32 Dword FIFO memory
*)
IF rst THEN
	(* asynchronous reset for the fifo *)
	NW := 0;
	NR := 0;
	Dout := 0;
	empty := TRUE;
	full := FALSE;
ELSIF WR AND E AND NOT full THEN
	(* write action *)
	fifo[NW] := Din;
	IF NW = top THEN NW := 0; ELSE NW := NW + 1; END_IF;
	full := NW = NR;
	empty := FALSE;
ELSIF NOT WR AND E AND NOT empty THEN
	(* read from stack *)
	Dout := fifo[NR];
	IF NR = top THEN NR := 0; ELSE NR := NR + 1; END_IF;
	empty := NR = NW;
	full := FALSE;
END_IF;

(* revision history
hm		4. aug. 2006	rev 1.0
	original version

hm		19. feb 2008	rev 1.1
	performance improvements

*)
END_FUNCTION_BLOCK

(* POU Logic/memory/STACK_16, ST *)
FUNCTION_BLOCK STACK_16
VAR_INPUT
	Din : DWORD;
	RW : BOOL;
	E : BOOL;
	RST : BOOL;
END_VAR
VAR_OUTPUT
	Dout : DWORD := 0;
	empty : BOOL := TRUE;
	full : BOOL := FALSE;
END_VAR
VAR
	Stack : ARRAY[0..15] OF DWORD;
	N : INT := -1;
	top : INT := 15;
END_VAR

(*
	version 1.1	19 feb 2008
	programmer 	hugo
	tested by		tobias

16 Dword STACK memory
*)
IF rst THEN
	(* asynchronous reset for the fifo *)
	N := -1;
	Dout := 0;
	empty := TRUE;
	full := FALSE;
ELSIF RW AND E AND NOT full THEN
	(* write action *)
	N := N + 1;
	full := N = TOP;
	empty := FALSE;
	stack[N] := Din;
ELSIF NOT RW AND E AND NOT empty THEN
	(* read from stack *)
	Dout := stack[N];
	N := N -1;
	empty := N < 0;
	full := FALSE;
END_IF;


(* revision history
hm		4. aug. 2006	rev 1.0
	original version

hm		19. feb 2008	rev 1.1
	performance improvements

*)
END_FUNCTION_BLOCK

(* POU Logic/memory/STACK_32, ST *)
FUNCTION_BLOCK STACK_32
VAR_INPUT
	Din : DWORD;
	RW : BOOL;
	E : BOOL;
	RST : BOOL;
END_VAR
VAR_OUTPUT
	Dout : DWORD := 0;
	empty : BOOL := TRUE;
	full : BOOL := FALSE;
END_VAR
VAR
	Stack : ARRAY[0..31] OF DWORD;
	N : INT := -1;
	top : INT := 31;
END_VAR

(*
	version 1.1	19. feb 2008
	programmer 	hugo
	tested by		tobias

32 Dword STACK memory
*)
IF rst THEN
	(* asynchronous reset for the fifo *)
	N := -1;
	Dout := 0;
	empty := TRUE;
	full := FALSE;
ELSIF RW AND E AND NOT full THEN
	(* write action *)
	N := N + 1;
	full := N = TOP;
	empty := FALSE;
	stack[N] := Din;
ELSIF NOT RW AND E AND NOT empty THEN
	(* read from stack *)
	Dout := stack[N];
	N := N -1;
	empty := N < 0;
	full := FALSE;
END_IF;


(* revision history
hm		4. aug. 2006	rev 1.0
	original version

hm		19. feb 2008	rev 1.1
	performance improvements

*)
END_FUNCTION_BLOCK

(* POU Logic/Others/matrix, ST *)
FUNCTION_BLOCK matrix
VAR_INPUT
	x1, x2, x3, x4, X5 : BOOL;
END_VAR
VAR_INPUT CONSTANT
	Release : BOOL;
END_VAR
VAR_OUTPUT
	code : BYTE;
	TP : BOOL;
	y1: BOOL := TRUE;
	y2, y3, y4 : BOOL;
END_VAR
VAR
	line : BYTE := 1;
	X : ARRAY[1..4] OF BYTE; (* scan line inputs *)
	L : ARRAY[1..4] OF BYTE; (* scan line status *)
	i: INT;
	temp: BYTE;
END_VAR

(*
version 1.2	23 dec 2007
programmer 	hugo
tested by		tobias

MATRIX is a matrix keyboard encoder for 4 rows and up to 5 columns.
matrix can send a code while a key is pressed and it sends another code while a key is released when the setup variable 'release' is set to true.
the setup variable release is false the code is only sent when the key is pressed.
the output byte holds the 5 columns in the lowest bits 0..2  and the row number in bits 4..6, while bit 7 is true for a key pressed and false for a key released.

*)
TP := FALSE;
code := 0;

(* read scan lines *)
X[line].0 := X1;
X[line].1 := X2;
X[line].2 := X3;
X[line].3 := X4;
X[line].4 := X5;

(* compare for change *)
FOR i := 1 TO 4 DO
	IF X[i] <> L[i] THEN
		(* scan line information has changed code need to be found and generated *)
		temp := x[i] XOR L[i];
		IF temp.0 THEN
			code := 1;
			code.7 := X[i].0;
			L[i].0 := X[i].0;
		ELSIF temp.1 THEN
			code := 2;
			code.7 := X[i].1;
			L[i].1 := X[i].1;
		ELSIF temp.2 THEN
			code := 3;
			code.7 := X[i].2;
			L[i].2 := X[i].2;
		ELSIF temp.3 THEN
			code := 4;
			code.7 := X[i].3;
			L[i].3 := X[i].3;
		ELSIF temp.4 THEN
			code := 5;
			code.7 := X[i].4;
			L[i].4 := X[i].4;
		END_IF;
		TP := TRUE;
		Code.4 := Line.0;
		Code.5 := Line.1;
		Code.6 := Line.2;

		(* check if release codes need to be killed *)
		IF NOT release AND code < 127 THEN
			code := 0;
			TP := 0;
		END_IF;
		EXIT;
	END_IF;
END_FOR;

(* increment scan line every cycle *)
CASE line OF
	1 :	Line := 2;
		Y1 := FALSE; Y3 := FALSE; Y4 := FALSE; Y2 := TRUE;
	2 :	Line := 3;
		Y1 := FALSE; Y2 := FALSE; Y4 := FALSE; Y3 := TRUE;
	3 :	Line := 4;
		Y1 := FALSE; Y2 := FALSE; Y3 := FALSE; Y4 := TRUE;
	4 :	Line := 1;
		Y2 := FALSE; Y3 := FALSE; Y4 := FALSE; Y1 := TRUE;
END_CASE;

(* revision history
hm		10.6.2007	rev 1.0		
	original version 


hm		11.9.2007	rev 1.1		
	deleted unused variables k and old_code

hm		23.12.2007	rev 1.2
	added exit statement in for loop instead of i:=5

*)
END_FUNCTION_BLOCK

(* POU mathematical/functions/FT_avg, ST *)
FUNCTION_BLOCK FT_avg
VAR_INPUT
	in : REAL;
	en : BOOL;
	N : INT;
	rst : BOOL;
END_VAR
VAR_OUTPUT
	avg : REAL;
END_VAR
VAR
	buff : delay;
	i: INT;
	init : BOOL;
END_VAR

(*
version 1.1	7 jan 2007
programmer 	hugo
tested by		tobias

this function calculates the average over n samples from a sequential input
the input values are shifted into an N deep buffer and the avg of this buffer is diplayed at anytime on the output.
a rst will load the buffer with the current in value..

*)
(* limit n to a max of 32 because delay can do max 32 cycles *)
IF N > 32 THEN
	buff.n := 32;
ELSIF N < 0 THEN
	Buff.n := 0;
ELSE
	buff.n := N;
END_IF;

IF NOT init THEN
	FOR i := 1 TO N DO
		buff(in := in);
	END_FOR;
	avg := in;
	init := TRUE;
ELSIF rst THEN
	FOR i := 1 TO N DO
		buff(in := in);
	END_FOR;
	avg := in;
ELSIF en THEN
	buff(in := in);
	avg := avg + (in - buff.out)/N;
END_IF;

(* revision history

hm	7.1.2007	rev 1.1
	chaged rst logic to load the buffer with the actual input value instead of 0.
	added en input to allow better control of signal flow
	added init to load the buffer with in at startup to avoid rampup at beginning.
	deleted unused variable cnt.
*)
END_FUNCTION_BLOCK

(* POU mathematical/functions/FT_min_max, ST *)
FUNCTION_BLOCK FT_min_max
VAR_INPUT
	in : REAL;
	rst : BOOL;
END_VAR
VAR_OUTPUT
	mx : REAL;
	mn : REAL;
END_VAR
VAR
	init: BOOL;
END_VAR

(*
version 1.0	1 sep 2006
programmer 	hugo
tested by		tobias

this function block stores the min and max value of an input signal.
when rst is true the mn and mx outputs are set to the in value.
when a rst is never active the function autoresets to the in value at startup.
since the input might not be present at first cycle the mn and mx are set during second cycle.

*)
IF rst OR NOT init THEN
	mn := in;
	mx := in;
	init := 1;
ELSIF in < mn THEN mn := in;
ELSIF in > mx THEN mx := in;
END_IF;
END_FUNCTION_BLOCK

(* POU Time&Date/Ltime, ST *)
FUNCTION_BLOCK Ltime
VAR_INPUT
	UTC : DT;
	dst_enable : BOOL;
	time_zone_offset : INT;
END_VAR
VAR_OUTPUT
	local_DT : DT;
	DST_on : BOOL;
	wday : INT;
END_VAR
VAR
	tx: TIME;
END_VAR

(*

version 1.6	8 dec 2007
programmer 	oscat
tested by		tobias

ltime is a real time clock that uses the system rtc as utc time and calculates and given time zone.
the utc time is supplied on the input UTC.
according to the input variable time_zone_offset when the input dst_enable is true,
the dst on and off times are calculated by a formula for any given year and the time is advanced and reset by one hour
at 02:00 and 03:00 for the last sunday of march and last sunday of october.
the code is high performance and the rtc counts every second.
if more then one time zone is needed by the systen the clock can be started many times by placing more then one function block.

execution time on wago 750-841 = 20 us 
 
*)
tx := DWORD_TO_TIME(INT_TO_DWORD(ABS(time_zone_offset))* 3600000);
DST_ON := DST(UTC) AND dst_enable;
IF DST_ON THEN
	IF time_zone_offset < 0 THEN local_DT := UTC - tx + t#1h; ELSE local_DT := UTC + tx + t#1h; END_IF;
ELSE
	IF time_zone_offset < 0 THEN local_DT := UTC - tx; ELSE local_DT := UTC + tx; END_IF;
END_IF;
wday := weekday(DT_TO_DATE(local_DT));


(* revision history

hm 2.10.2006	rev 1.1
	corrected an error where dst would be delayed by 0.1second

hm 17.1.2007	rev 1.2
	added utc input instead of internal sysrtcgettime because this would only work on wago.
	dst_enable would not be checked before dst would be enabled.

hm 18.3.2007	rev 1.3
	changed code, dst would not work during first cycle.

hm 24.10.2007	rev 1.4
	changed code because the execution every 100ms can cause major problems if the supplied time was not correct at start.
	use of new dst function

hm 12. nov 2007	rev 1.5
		changed Type of time_zone_offset from time to int to allow for time zones with negative offset

8 dec 2007		rev 1.6
	corrected a problem with time_zone_offset
*)
END_FUNCTION_BLOCK

(* POU XTEST/Performance Test/fc_list, ST *)
FUNCTION_BLOCK fc_list
VAR_INPUT
	num : INT;
	check : BOOL;
	arr : ARRAY[0..63] OF BYTE;
	rar : ARRAY[0..63] OF REAL := 134653,12534,1234,134,12,123,3,7,33,55,200,300,700,2,5,3,7657,2345,4,65,88,435,23465346,0,0,0,5,5,5,9,9,9,300,200,100,50,36,25,20,28,27,25,4567,347,3476,4357,468,3865,6,356,4564,55,3457,1,4,7,9,13,14,15,16,17,18,55;
	ra1 : ARRAY[0..4] OF REAL := 5,3,4,1,2;
END_VAR
VAR
	ARRp: ARRAY [1..20,0..1] OF REAL :=  -10,-0.53, 10,0.53, 100,88.3, 200,122.2;
	ARRq: ARRAY [1..5,0..1] OF REAL :=  -10,-0.53, 10,0.53, 100,88.3, 200,122.2;
	va,vb : vector_3;
	ptn : INT := 4;
	X : REAL := 1000;
	Y: INT := 1000;
	ptx : POINTER TO DWORD;
END_VAR
ptx := ADR(X);
IF num < 10 THEN
	CASE num OF
	0 :	IF check THEN RETURN; ELSE RETURN; END_IF;
	1 : IF check THEN RETURN; ELSE Air_density(20,101525,0.5); END_IF;
 	2 : IF check THEN RETURN; ELSE Air_enthalpy(20,50); END_IF;
	3 : IF check THEN RETURN; ELSE dew_con(50,20); END_IF;
	4 : IF check THEN RETURN; ELSE dew_temp(50,20); END_IF;
	5 : IF check THEN RETURN; ELSE Heat_index(20,50); END_IF;
	6 : IF check THEN RETURN; ELSE SDD(20,TRUE); END_IF;
	7 : IF check THEN RETURN; ELSE water_CP(20); END_IF;
	8 : IF check THEN RETURN; ELSE Water_density(20,TRUE); END_IF;
	9 : IF check THEN RETURN; ELSE water_enthalpy(20); END_IF;
	END_CASE;
ELSIF num < 20 THEN
	CASE num OF
	10 : IF check THEN RETURN; ELSE WCT(-10,50); END_IF;
	11 : IF check THEN RETURN; ELSE dead_band(20,5); END_IF;
	12 : IF check THEN RETURN; ELSE dead_zone(20,5); END_IF;
	13 : IF check THEN RETURN; ELSE C_to_F(10); END_IF;
	14 : IF check THEN RETURN; ELSE C_to_K(3.2); END_IF;
	15 : IF check THEN RETURN; ELSE F_to_C(10.0); END_IF;
	16 : IF check THEN RETURN; ELSE F_to_OM(200); END_IF;
	17 : IF check THEN RETURN; ELSE F_to_PT(200); END_IF;
	18 : IF check THEN RETURN; ELSE K_to_C(20); END_IF;
	19 : IF check THEN RETURN; ELSE KMH_TO_MS(10.0); END_IF;
	END_CASE;
ELSIF num < 30 THEN
	CASE num OF
	20 : IF check THEN RETURN; ELSE MS_TO_KMH(20); END_IF;
	21 : IF check THEN RETURN; ELSE OM_to_F(120); END_IF;
	22 : IF check THEN RETURN; ELSE PT_to_F(T#200ms); END_IF;
	23 : IF check THEN RETURN; ELSE T_PLC_MS(); END_IF;
	24 : IF check THEN RETURN; ELSE T_PLC_US(); END_IF;
	25 : IF check THEN RETURN; ELSE multi_in(1,2,3,4,5,6,0); END_IF;
	26 : IF check THEN RETURN; ELSE Res_NI(20,10000); END_IF;
	27 : IF check THEN RETURN; ELSE Res_PT(20,10000); END_IF;
	28 : IF check THEN RETURN; ELSE Res_SI(20,10000,20); END_IF;
	29 : IF check THEN RETURN; ELSE Sensor_Int(10,0.1,1000000,1); END_IF;
	END_CASE;
ELSIF num < 40 THEN
	CASE num OF
	30 : IF check THEN RETURN; ELSE Temp_NI(1233,1000); END_IF;
	31 : IF check THEN RETURN; ELSE Temp_PT(1233,1000); END_IF;
	32 : IF check THEN RETURN; ELSE Temp_SI(1233,1000,20); END_IF;
	33 : IF check THEN RETURN; ELSE AIN(1000,12,15,10.0,100.0); END_IF;
	34 : IF check THEN RETURN; ELSE Aout(10.0,12,15,10.0,100.0); END_IF;
	35 : IF check THEN RETURN; ELSE MIX(100,200,0.5); END_IF;
	36 : IF check THEN RETURN; ELSE MUX_R2(10.0,10.0,TRUE); END_IF;
	37 : IF check THEN RETURN; ELSE MUX_R4(10.0,10.0,10.0,10.0,TRUE,TRUE); END_IF;
	38 : IF check THEN RETURN; ELSE Offset(10.0,TRUE,TRUE,TRUE,TRUE,TRUE,10.0,10.0,10.0,10.0,1.0); END_IF;
	39 : IF check THEN RETURN; ELSE Offset2(10.0,TRUE,TRUE,TRUE,TRUE,TRUE,10.0,10.0,10.0,10.0,1.0); END_IF;
	END_CASE;
ELSIF num < 50 THEN
	CASE num OF
	40 : IF check THEN RETURN; ELSE Override(1,2,3,TRUE,TRUE,TRUE); END_IF;
	41 : IF check THEN RETURN; ELSE scale_B2(100,100,10.0,10.0,10.0,10.0,10.0,10.0); END_IF;
	42 : IF check THEN RETURN; ELSE scale_B4(100,100,100,100,10.0,10.0,10.0,10.0,10.0,10.0,10.0,10.0,10.0,10.0); END_IF;
	43 : IF check THEN RETURN; ELSE scale_B8(100,100,100,100,100,100,100,100,10.0,10.0,10.0,10.0,10.0,10.0,10.0,10.0,10.0,10.0,10.0,10.0,10.0,10.0,10.0,10.0,10.0,10.0); END_IF;
	44 : IF check THEN RETURN; ELSE scale_X2(TRUE,TRUE,10.0,10.0,10.0,10.0,10.0,10.0); END_IF;
	45 : IF check THEN RETURN; ELSE scale_X4(TRUE,TRUE,TRUE,TRUE,10.0,10.0,10.0,10.0,10.0,10.0,10.0,10.0,10.0,10.0); END_IF;
	46 : IF check THEN RETURN; ELSE scale_X8(TRUE,TRUE,TRUE,TRUE,TRUE,TRUE,TRUE,TRUE,10.0,10.0,10.0,10.0,10.0,10.0,10.0,10.0,10.0,10.0,10.0,10.0,10.0,10.0,10.0,10.0,10.0,10.0); END_IF;
	47 : IF check THEN RETURN; ELSE stair(10.0,1.0); END_IF;
	48 : IF check THEN RETURN; ELSE BCD_TO_INT(44); END_IF;
	49 : IF check THEN RETURN; ELSE Bit_Count(100); END_IF;
	END_CASE;
ELSIF num < 60 THEN
	CASE num OF
	50 : IF check THEN RETURN; ELSE Bit_of_Dword(1000,2); END_IF;
	51 : IF check THEN RETURN; ELSE Byte_of_bit(TRUE,TRUE,TRUE,TRUE,TRUE,TRUE,TRUE,TRUE); END_IF;
	52 : IF check THEN RETURN; ELSE Byte_of_Dword(1000,2); END_IF;
	53 : IF check THEN RETURN; ELSE check_parity(1000,TRUE); END_IF;
	54 : IF check THEN RETURN; ELSE DWord_of_Byte(100,100,100,100); END_IF;
	55 : IF check THEN RETURN; ELSE INT_TO_BCD(123); END_IF;
	56 : IF check THEN RETURN; ELSE mux_2(TRUE,TRUE,TRUE); END_IF;
	57 : IF check THEN RETURN; ELSE mux_4(TRUE,TRUE,TRUE,TRUE,TRUE,TRUE); END_IF;
	58 : IF check THEN RETURN; ELSE parity(2000); END_IF;
	59 : IF check THEN RETURN; ELSE reverse(123); END_IF;
	END_CASE;
ELSIF num < 70 THEN
	CASE num OF
	60 : IF check THEN RETURN; ELSE SHL1(123,1); END_IF;
	61 : IF check THEN RETURN; ELSE SHR1(123,1); END_IF;
	62 : IF check THEN RETURN; ELSE Word_of_Byte(100,100); END_IF;
	63 : IF check THEN RETURN; ELSE Word_of_Dword(2000,1); END_IF;
	64 : IF check THEN RETURN; ELSE CRC_CHECK(ADR(arr),SIZEOF(arr),2000,FALSE); END_IF;
	65 : IF check THEN RETURN; ELSE CRC_GEN(ADR(arr),SIZEOF(Arr),2000,FALSE, 0,0,FALSE, FALSE); END_IF;
	66 : IF check THEN RETURN; ELSE _array_init(ADR(rar),SIZEOF(rar),10.0); END_IF;
	67 : IF check THEN RETURN; ELSE _array_median(ADR(rar),SIZEOF(rar)); END_IF;
	68 : IF check THEN RETURN; ELSE _array_sort(ADR(rar),SIZEOF(rar)); END_IF;
	69 : IF check THEN RETURN; ELSE array_avg(ADR(rar),SIZEOF(rar)); END_IF;
	END_CASE;
ELSIF num < 80 THEN
	CASE num OF
	70 : IF check THEN RETURN; ELSE array_max(ADR(rar),SIZEOF(rar)); END_IF;
	71 : IF check THEN RETURN; ELSE array_min(ADR(rar),SIZEOF(rar)); END_IF;
	72 : IF check THEN RETURN; ELSE array_sdv(ADR(rar),SIZEOF(rar)); END_IF;
	73 : IF check THEN RETURN; ELSE array_spr(ADR(rar),SIZEOF(rar)); END_IF;
	74 : IF check THEN RETURN; ELSE array_sum(ADR(rar),SIZEOF(rar)); END_IF;
	75 : IF check THEN RETURN; ELSE array_trend(ADR(ra1),SIZEOF(ra1)); END_IF;
	76 : IF check THEN RETURN; ELSE array_var(ADR(rar),SIZEOF(rar)); END_IF;
	77 : IF check THEN RETURN; ELSE F_lin(10.0,10.0,10.0); END_IF;
	78 : IF check THEN RETURN; ELSE F_Lin2(10.0,10.0,10.0,10.0,10.0); END_IF;
	79 : IF check THEN RETURN; ELSE F_power(10.0,10.0,10.0); END_IF;
	END_CASE;
ELSIF num < 90 THEN
	CASE num OF
	80 : IF check THEN RETURN; ELSE F_quad(10.0,10.0,10.0,10.0); END_IF;
	81 : IF check THEN RETURN; ELSE LINEAR_INT(X, ARRp, ptn); END_IF;
	82 : IF check THEN RETURN; ELSE POLYNOM_INT(x, arrq, ptn); END_IF;
	83 : IF check THEN RETURN; ELSE circle_A(10,10); END_IF;
	84 : IF check THEN RETURN; ELSE circle_C(10,10); END_IF;
	85 : IF check THEN RETURN; ELSE cone_V(10,10); END_IF;
	86 : IF check THEN RETURN; ELSE ellipse_A(10,10); END_IF;
	87 : IF check THEN RETURN; ELSE ellipse_C(10,10); END_IF;
	88 : IF check THEN RETURN; ELSE sphere_V(10); END_IF;
	89 : IF check THEN RETURN; ELSE triangle_A(1,2,3,4); END_IF;
	END_CASE;
ELSIF num < 100 THEN
	CASE num OF
	90 : IF check THEN RETURN; ELSE V3_ABS(va); END_IF;
	91 : IF check THEN RETURN; ELSE V3_ADD(va,vb); END_IF;
	92 : IF check THEN RETURN; ELSE V3_ANG(va,vb); END_IF;
	93 : IF check THEN RETURN; ELSE V3_DPRO(va,vb); END_IF;
	94 : IF check THEN RETURN; ELSE V3_NORM(va); END_IF;
	95 : IF check THEN RETURN; ELSE V3_NUL(va); END_IF;
	96 : IF check THEN RETURN; ELSE V3_PAR(va,vb); END_IF;
	97 : IF check THEN RETURN; ELSE V3_REV(va); END_IF;
	98 : IF check THEN RETURN; ELSE V3_SMUL(va,3); END_IF;
	99 : IF check THEN RETURN; ELSE V3_SUB(va,vb); END_IF;
	END_CASE;
ELSIF num < 110 THEN
	CASE num OF
	100 : IF check THEN RETURN; ELSE V3_XANG(va); END_IF;
	101 : IF check THEN RETURN; ELSE V3_XPRO(va,vb); END_IF;
	102 : IF check THEN RETURN; ELSE V3_YANG(va); END_IF;
	103 : IF check THEN RETURN; ELSE V3_ZANG(va); END_IF;
	104 : IF check THEN RETURN; ELSE acosH(5); END_IF;
	105 : IF check THEN RETURN; ELSE acotH(5); END_IF;
	106 : IF check THEN RETURN; ELSE asinH(5); END_IF;
	107 : IF check THEN RETURN; ELSE atanH(0.5); END_IF;
	108 : IF check THEN RETURN; ELSE ceil(1.3); END_IF;
	109 : IF check THEN RETURN; ELSE cosH(5); END_IF;
	END_CASE;
ELSIF num < 120 THEN
	CASE num OF
	110 : IF check THEN RETURN; ELSE cotH(5); END_IF;
	111 : IF check THEN RETURN; ELSE deg(0.5); END_IF;
	112 : IF check THEN RETURN; ELSE differ(10.0,20.0,15.0); END_IF;
	113 : IF check THEN RETURN; ELSE even(2); END_IF;
	114 : IF check THEN RETURN; ELSE exp10(3); END_IF;
	115 : IF check THEN RETURN; ELSE expn(23,3); END_IF;
	116 : IF check THEN RETURN; ELSE fact(5); END_IF;
	117 : IF check THEN RETURN; ELSE floor(2.3); END_IF;
	118 : IF check THEN RETURN; ELSE fract(2.3); END_IF;
	119 : IF check THEN RETURN; ELSE gamma(34); END_IF;
	END_CASE;
ELSIF num < 130 THEN
	CASE num OF
	120 : IF check THEN RETURN; ELSE inc(1,2,3); END_IF;
	121 : IF check THEN RETURN; ELSE Langevin(3); END_IF;
	122 : IF check THEN RETURN; ELSE max3(10.0,20.0,15.0); END_IF;
	123 : IF check THEN RETURN; ELSE mid3(10.0,20.0,15.0); END_IF;
	124 : IF check THEN RETURN; ELSE min3(10.0,20.0,15.0); END_IF;
	125 : IF check THEN RETURN; ELSE modR(10.0,2.0); END_IF;
	126 : IF check THEN RETURN; ELSE MUL_ADD(10.0,10.0,10.0); END_IF;
	127 : IF check THEN RETURN; ELSE neg(3); END_IF;
	128 : IF check THEN RETURN; ELSE Rad(0.5); END_IF;
	129 : IF check THEN RETURN; ELSE RDM(0); END_IF;
	END_CASE;
ELSIF num < 140 THEN
	CASE num OF
	130 : IF check THEN RETURN; ELSE round(10.9,3); END_IF;
	131 : IF check THEN RETURN; ELSE sgn(3); END_IF;
	132 : IF check THEN RETURN; ELSE sigmoid(10.4); END_IF;
	133 : IF check THEN RETURN; ELSE sign_I(3); END_IF;
	134 : IF check THEN RETURN; ELSE sign_R(4.0); END_IF;
	135 : IF check THEN RETURN; ELSE sinH(0.5); END_IF;
	136 : IF check THEN RETURN; ELSE sqrtn(34,3); END_IF;
	137 : IF check THEN RETURN; ELSE tanH(0.5); END_IF;
	138 : IF check THEN RETURN; ELSE window(1,2,3); END_IF;
	139 : IF check THEN RETURN; ELSE window2(1,2,3); END_IF;
	END_CASE;
ELSIF num < 150 THEN
	CASE num OF
	140 : IF check THEN RETURN; ELSE BYTE_TO_STRB(100); END_IF;
	141 : IF check THEN RETURN; ELSE BYTE_TO_STRH(100); END_IF;
	142 : IF check THEN RETURN; ELSE CHR(22); END_IF;
	143 : IF check THEN RETURN; ELSE DWORD_TO_STRB(2000); END_IF;
	144 : IF check THEN RETURN; ELSE DWORD_TO_STRH(2000); END_IF;
	145 : IF check THEN RETURN; ELSE DWORD_To_STRF(2000,3); END_IF;
	146 : IF check THEN RETURN; ELSE exec('3+4'); END_IF;
	147 : IF check THEN RETURN; ELSE find_nonum('jhgfu'); END_IF;
	148 : IF check THEN RETURN; ELSE find_Num('jhgfu'); END_IF;
	149 : IF check THEN RETURN; ELSE FindB('jhgfu','hh'); END_IF;
	END_CASE;
ELSIF num < 160 THEN
	CASE num OF
	150 : IF check THEN RETURN; ELSE findB_nonum('jhgfu'); END_IF;
	151 : IF check THEN RETURN; ELSE findB_Num('jhgfu'); END_IF;
	152 : IF check THEN RETURN; ELSE HEX_TO_DWORD('4444'); END_IF;
	153 : IF check THEN RETURN; ELSE lowercase('Sepp faehrt im Taxi nach Kalkutta'); END_IF;
	154 : IF check THEN RETURN; ELSE Real_To_StrF(10.345,4); END_IF;
	155 : IF check THEN RETURN; ELSE trim('fvr54tg h'); END_IF;
	156 : IF check THEN RETURN; ELSE uppercase('Sepp faehrt im Taxi nach Kalkutta'); END_IF;
	157 : IF check THEN RETURN; ELSE date_add(d#2007-8-12,1,1,1,1); END_IF;
	158 : IF check THEN RETURN; ELSE day_of_date(d#2007-1-1); END_IF;
	159 : IF check THEN RETURN; ELSE day_of_month(d#2007-8-12); END_IF;
	END_CASE;
ELSIF num < 170 THEN
	CASE num OF
	160 : IF check THEN RETURN; ELSE day_of_year(d#2007-8-12); END_IF;
	161 : IF check THEN RETURN; ELSE day_to_time(23); END_IF;
	162 : IF check THEN RETURN; ELSE days_delta(d#2007-8-12,d#2007-8-12); END_IF;
	163 : IF check THEN RETURN; ELSE DST(dt#2007-8-12-12:00); END_IF;
	164 : IF check THEN RETURN; ELSE easter(2007); END_IF;
	165 : IF check THEN RETURN; ELSE hour(TOD#12:00); END_IF;
	166 : IF check THEN RETURN; ELSE hour_to_time(3.14); END_IF;
	167 : IF check THEN RETURN; ELSE hour_to_tod(3.14); END_IF;
	168 : IF check THEN RETURN; ELSE leap_of_Date(d#2007-8-12); END_IF;
	169 : IF check THEN RETURN; ELSE leap_year(2007); END_IF;
	END_CASE;
ELSIF num < 180 THEN
	CASE num OF
	170 : IF check THEN RETURN; ELSE dew_rh(20,1); END_IF;
	171 : IF check THEN RETURN; ELSE local_time(dt#2007-8-12-12:00,1,TRUE); END_IF;
	172 : IF check THEN RETURN; ELSE Ltime_to_UTC(dt#2007-8-12-12:00,TRUE,1); END_IF;
	173 : IF check THEN RETURN; ELSE minute(TOD#12:00); END_IF;
	174 : IF check THEN RETURN; ELSE minute_to_time(3.14); END_IF;
	175 : IF check THEN RETURN; ELSE month(d#2007-8-12); END_IF;
	176 : IF check THEN RETURN; ELSE multime(t#1h,3.2); END_IF;
	177 : IF check THEN RETURN; ELSE period(d#2007-9-1,D#2007-10-1,D#2007-11-1); END_IF;
	178 : IF check THEN RETURN; ELSE second(tod#12:00); END_IF;
	179 : IF check THEN RETURN; ELSE second_to_time(3.14); END_IF;
	END_CASE;
ELSIF num < 190 THEN
	CASE num OF
	180 : IF check THEN RETURN; ELSE set_Date(2007,12,12); END_IF;
	181 : IF check THEN RETURN; ELSE set_DT(2007,12,12,1,1,1); END_IF;
	182 : IF check THEN RETURN; ELSE set_Tod(12,13,3.23); END_IF;
	183 : IF check THEN RETURN; ELSE weekday(d#2007-8-12); END_IF;
	184 : IF check THEN RETURN; ELSE work_week(d#2007-8-12); END_IF;
	185 : IF check THEN RETURN; ELSE year_begin(2007); END_IF;
	186 : IF check THEN RETURN; ELSE year(d#2038-7-24); END_IF;
	187 : IF check THEN RETURN; ELSE fib(29); END_IF;
	188 : IF check THEN RETURN; ELSE RETURN; END_IF;
	189 : IF check THEN RETURN; ELSE RETURN; END_IF;
	END_CASE;
ELSIF num < 200 THEN
	CASE num OF
	190 : IF check THEN RETURN; ELSE X := X / 2; END_IF;
	191 : IF check THEN RETURN; ELSE Y := Y / 2; END_IF;
	192 : IF check THEN RETURN; ELSE ptx^ := ROL(ROR(ptx^,23)-1,23); END_IF;
	193 : IF check THEN RETURN; ELSE Y := SHR(Y,1); END_IF;
	194 : IF check THEN RETURN; ELSE X := X * 2; END_IF;
	195 : IF check THEN RETURN; ELSE Y := Y * 2; END_IF;
	196 : IF check THEN RETURN; ELSE Y := SHL(Y,1); END_IF;
	197 : IF check THEN RETURN; ELSE RETURN; END_IF;
	198 : IF check THEN RETURN; ELSE RETURN; END_IF;
	199 : IF check THEN RETURN; ELSE RETURN; END_IF;
	END_CASE;
END_IF;
END_FUNCTION_BLOCK

(* POU Building/HLK/Heat_index, ST *)
FUNCTION Heat_index : REAL
VAR_INPUT
	T : REAL;
	RH : REAL;
END_VAR
VAR
	RH2 : REAL;
	T2 : REAL;
END_VAR

(*
version 1.2	2 dec 2007
programmer 	hugo
tested by		tobias

this function calculates the heat index temperature depending on external temperature and Relative humidity

*)
IF RH < 20 OR T < 20 THEN
	Heat_index := T;
ELSE
	RH2 := RH * RH;
	T := C_to_F(T);
	T2 := T * T;
	Heat_index := -42.379 + 2.04901523 * T - 6.83783E-3 * T2
			+ RH * (10.1433127 - 0.22475541 * T + 1.22874E-3 * T2)
			+ RH2 * (8.5282E-4 * T - 5.481717E-2 - 1.99E-6 * T2);
	Heat_index := F_to_C(Heat_index);
END_IF;

(* revision history

hm 27.2.2007		rev 1.1
	deleted unused variables rh3 and T3

hm	2.12.2007		rev 1.2
	changed code for better performance
*)
END_FUNCTION

(* POU Building/HLK/WCT, ST *)
FUNCTION WCT : REAL
VAR_INPUT
	T : REAL;
	V : REAL;
END_VAR
VAR
END_VAR

(*
version 1.1	7 dec 2007
programmer 	hugo
tested by		tobias

this function calculates the wind chill temperature

*)
IF V < 5 OR T > 10 THEN
	WCT := T;
ELSE
	WCT := 13.12 + 0.6215 * T +(0.3965 * T - 11.37) * EXP(LN(v) * 0.16);
END_IF;


(* revision history
hm		7 feb 2007
	original version

hm		7 dec 2007
	changed code for better performance

*)
END_FUNCTION

(* POU engineering/conversion/K_to_C, ST *)
FUNCTION K_to_C : REAL
VAR_INPUT
	Kelvin : REAL;
END_VAR
VAR
END_VAR

(*
version 1.0	4 dec 2006
programmer 	hugo
tested by		tobias

this function converts kelvin to celsius
*)
K_to_C := Kelvin + 273.15;
END_FUNCTION

(* POU engineering/conversion/KMH_TO_MS, ST *)
FUNCTION KMH_TO_MS : REAL
VAR_INPUT
	kmh : REAL;
END_VAR
VAR
END_VAR

(*
version 1.1	6 jan 2007
programmer 	hugo
tested by		tobias

this function converts velocities from Kilometers / hour to Meters / Second

*)
KMH_TO_MS := kmh * 0.2777777777777;

(* revision history
hm	4. feb 2007		rev 1.0
	original version

hm	6. jan 2008		rev 1.1
	improved performance

*)
END_FUNCTION

(* POU engineering/conversion/MS_TO_KMH, ST *)
FUNCTION MS_TO_KMH : REAL
VAR_INPUT
	ms : REAL;
END_VAR
VAR
END_VAR

(*
version 1.0	4 Feb 2007
programmer 	hugo
tested by		tobias

this function converts velocities from Meters / Second to Kilometers / hour.

*)
MS_TO_KMH := ms * 3.6;
END_FUNCTION

(* POU engineering/conversion/OM_to_F, ST *)
FUNCTION OM_to_F : REAL
VAR_INPUT
	OM : REAL;
END_VAR
VAR
END_VAR

(*
version 1.0	22 jan 2007
programmer 	hugo
tested by		tobias

this function converts Omega F to frequency
F = OM / (2*PI)
*)
OM_to_F := OM / PI2;
END_FUNCTION

(* POU engineering/conversion/PT_to_F, ST *)
FUNCTION PT_to_F : REAL
VAR_INPUT
	PT : TIME;
END_VAR
VAR
END_VAR

(*
version 1.0	4 aug 2006
programmer 	hugo
tested by		tobias

this function converts periode time to frequency
*)
PT_to_F := 1000/DWORD_TO_REAL(TIME_TO_DWORD(PT));
END_FUNCTION

(* POU engineering/sensor/Res_PT, ST *)
FUNCTION Res_PT : REAL
VAR_INPUT
	T : REAL;
	R0 : REAL;
END_VAR
VAR CONSTANT
	A : REAL := 3.90802E-3 ;
	B : REAL := -5.802E-7;
	C : REAL := -4.27350E-12;
END_VAR
VAR
	T2: REAL;
END_VAR

(*
version 1.2	2 dec 2007
programmer 	hugo
tested by		tobias


this function returs the resistance for a platinum sensor for a temperature range from -200..+850 °C *)
T2 := T * T;
IF T >= 0 THEN
	Res_PT := R0 * ( 1 + A*T + B*T2);
ELSE
	Res_PT := R0 * ( 1 + A*T + B*T2 + C*(T-100)*T2*T);
END_IF;

(* revision history
hm	4. aug. 2006	rev 1.1
	original version

hm	2. dec 2007		rev 1.2
	changed code for better performance

*)


(*
 Auszug aus DIN 43760 für Pt100

°C		R		°C		R		°C	R			°C		R			°C		R			°C		R

-200 	18,49 	-100 	60,25 	0 	100,00 	100 	138,50 	200 	175,84 	300 	212,02
-195 	20,65 	-95 	62,28 	5 	101,95 	105 	140,39 	205 	177,68 	305 	213,80
-190 	22,80 	-90 	64,30 	10 	103,90 	110 	142,29 	210 	179,51 	310 	215,57
-185 	24,94 	-85 	66,31 	15 	105,85 	115 	144,17 	215 	181,34 	315 	217,35
-180 	27,08 	-80 	68,33 	20 	107,79 	120 	146,06 	220 	183,17 	320 	219,12
-175 	29,20 	-75 	70,33 	25 	109,73 	125 	147,94 	225 	184,99 	325 	220,88
-170 	31,32 	-70 	72,33 	30 	111,67 	130 	149,82 	230 	186,82 	330 	222,65
-165 	33,43 	-65 	74,33 	35 	113,61 	135 	151,70 	235 	188,63 	335 	224,41
-160 	35,33 	-60 	76,33 	40 	115,54 	140 	153,58 	240 	190,45 	340 	226,17
-155 	37,63 	-55 	78,32 	45 	117,47 	145 	155,45 	245 	192,26 	345 	227,92
-150 	39,71 	-50 	80,31 	50 	119,40 	150 	157,31 	250 	194,07 	350 	229,67
-145 	41,79 	-45 	82,29 	55 	121,32 	155 	159,18 	255 	195,88 	355 	231,42
-140 	43,87 	-40 	84,27 	60 	123,24 	160 	161,04 	260 	197,69 	360 	233,17
-135 	45,94 	-35 	86,25 	65 	125,16 	165 	162,90 	265 	199,49 	365 	234,91
-130 	48,00 	-30 	88,22 	70 	127,07 	170 	164,76 	270 	201,29 	370 	236,65
-125 	50,06 	-25 	90,19 	75 	128,98 	175 	166,61 	275 	203,08 	375 	238,39
-120 	52,11 	-20 	92,16 	80 	130,89 	180 	168,46 	280 	204,88 	380 	240,13
-115 	54,15 	-15 	94,12 	85 	132,80 	185 	170,31 	285 	206,67 	385 	241,86
-110 	56,19 	-10 	96,09 	90 	134,70 	190 	172,16 	290 	208,45 	390 	243,59
-105 	58,22 	-5 		98,04 	95 	136,60 	195 	174,00 	295 	210,24 	395 	245,31

*)
(*
revision history


*)
END_FUNCTION

(* POU engineering/sensor/Sensor_Int, ST *)
FUNCTION Sensor_Int : REAL
VAR_INPUT
	Voltage : REAL;
	Current : REAL;
	RP : REAL;
	RS : REAL;
END_VAR
VAR
	RG: REAL;
END_VAR

(*
version 1.2	2 dec 2007
programmer 	hugo
tested by		tobias

this function calculates the real resistance of a sensor RX given a parasitic resistor in parallel to the sensor and an additional serial resistor.
for example a parasitic parallel resistor for a PT100 can be ignored but a series resistor is the cable to the sensor.
for a humidity sensor, the parallel resistor is more dramatic and needs to be considered.
the function allows to consider a parallel and serial resistor at the same time.
with this function and known parasitic serial and parallel resistors the true resistance of the sensor can be calculated.

*)
IF current <> 0 THEN
	RG := voltage / current;
	Sensor_Int := RP * ( RG - RS) / ( RP + RS - RG);
END_IF;

(* revisaion history

hm 20.1.2007	rev 1.1
	deleted input R0 which was not needed.

hm	2. dec 2007	rev 1.2
	corrected an error in formula and improoved speed
*)
END_FUNCTION

(* POU engineering/sensor/Temp_PT, ST *)
FUNCTION Temp_PT : REAL
VAR_INPUT
	Res : REAL;
	R0 : REAL;
END_VAR
VAR CONSTANT
	A : REAL := 3.9083E-3 ;
	B : REAL := -5.775E-7;
	accuracy : REAL := 0.02;
END_VAR
VAR
	step: REAL := 50.0;
	X: REAL;
	Y: REAL;
	t1: REAL;
END_VAR

(*
version 1.5	5. jan 2008
programmer 	hugo
tested by		tobias

this function returs the temperature for a platinum sensor for a range from -200..+850 °C *)
X := A * R0;
Y := B * R0;
IF Res >= R0 THEN
	t1 := X*X-4*Y*(R0-Res);
	IF t1 < 0 THEN
		Temp_PT := 10000;
	ELSE
		Temp_PT := (-X + SQRT(t1)) / (2 * Y);
	END_IF;
ELSE
	(* since the formula cannot be solved this is a successive approximation *)
	Temp_PT := -100.0;
	WHILE step > accuracy DO
		(* test if result greater or less *)
		IF Res_PT(Temp_PT,R0) < res THEN Temp_PT := Temp_PT + step; ELSE Temp_PT := Temp_PT - step; END_IF;
		step := step * 0.5;
	END_WHILE;
END_IF;

(* revision history

rev 1.1 hm 24.1.2007	
	deleted unused variable C

rev 1.2 hm 10.9.2007
	reduced accuracy to 0.02 to shorten execution time

rev 1.3	hm	2. dec 2007
	changed code for better performance

rev	1.4	hm	23. dec 2007
	avoid a negative square root if input values are wrong

rev 1.5 hm	5. jan 2008
	replaced / 2 with * 0.5 for better performance
*)
END_FUNCTION

(* POU engineering/signal processing/MIX, ST *)
FUNCTION MIX : REAL
VAR_INPUT
	A, B : REAL;
	M : REAL;
END_VAR
VAR
END_VAR

(*
version 1.0	19 nov 2007
programmer 	hugo
tested by		tobias

MIX is an analog Mixer. The Output is (1-M)*A + M*B.

*)
MIX := (1-M)*A + M*B;

(* revision history
hm	19. Nov 2007		rev 1.0
	original version
*)
END_FUNCTION

(* POU engineering/signal processing/MUX_R2, ST *)
FUNCTION MUX_R2 : REAL
VAR_INPUT
	IN0 : REAL;
	IN1 : REAL;
	A : BOOL;
END_VAR
VAR
END_VAR

(*
version 1.0	19 jan 2007
programmer 	oscat
tested by		tobias

MUX_R2 is an analog Multiplexer.
one of 2 real inputs are selected and put through to out.
The Adress input A selects between 2 Real inputs IN0 and IN1, A=0 > In0, A=1 > in1.

*)
IF NOT A THEN
	MUX_R2 := IN0;
ELSE
	MUX_R2 := IN1;
END_IF;
END_FUNCTION

(* POU engineering/signal processing/MUX_R4, ST *)
FUNCTION MUX_R4 : REAL
VAR_INPUT
	IN0 : REAL;
	IN1 : REAL;
	IN2 : REAL;
	IN3 : REAL;
	A0 : BOOL;
	A1 : BOOL;
END_VAR
VAR
END_VAR

(*
version 1.0	19 jan 2007
programmer 	oscat
tested by		tobias

MUX_R4 is an analog Multiplexer.
one of 4 real inputs are selected and put through to out.
The Adress input A0 and A1 selects between the 4 Real inputs IN0.. IN1.

*)
IF NOT A0 AND NOT A1 THEN
	MUX_R4 := IN0;
ELSIF A0 AND NOT a1 THEN
	MUX_R4 := IN1;
ELSIF NOT A0 AND A1 THEN
	MUX_R4 := IN2;
ELSE
	MUX_R4 := IN3;
END_IF;
END_FUNCTION

(* POU engineering/signal processing/Offset2, ST *)
FUNCTION Offset2 : REAL
VAR_INPUT
	X : REAL;
	O1, O2, O3, O4 : BOOL;
	D : BOOL;
END_VAR
VAR_INPUT CONSTANT
	Offset_1 : REAL;
	Offset_2 : REAL;
	Offset_3 : REAL;
	Offset_4 : REAL;
	default : REAL;
END_VAR

(*
version 1.0	12 jan 2007
programmer 	oscat
tested by		tobias

The Function offset adds offsets to an analog signal depending on digital inputs.
one offset can be added at the same time, if more then one input is true, the one with the highest number (o1 .. o4) will be used.
The input D will select a default value instead of X for input.

*) 
IF D THEN Offset2 := default; ELSE Offset2 := X; END_IF;
IF O4 THEN Offset2 := Offset2 + offset_4;
ELSIF O3 THEN Offset2 := Offset2 + offset_3;
ELSIF O2 THEN Offset2 := Offset2 + offset_2;
ELSIF O1 THEN Offset2 := Offset2 + offset_1;
END_IF;
END_FUNCTION

(* POU engineering/signal processing/Override, ST *)
FUNCTION Override : REAL
VAR_INPUT
	X1, X2, X3 : REAL;
	E1 : BOOL;
	E2 : BOOL;
	E3 : BOOL;
END_VAR
VAR
END_VAR

(*
version 1.0	4 nov 2007
programmer 	oscat
tested by	tobias

MAXR deliveres the maximum absolute value of the 3 inputs X1, X2 and X3.
with the inputs E1, E2 and E3 each of the 3 inputs can be turned on or off, while the default for these 3 inputs is true.

*) 
IF E1 THEN Override := X1; END_IF;
IF E2 AND ABS(x2) > ABS(Override) THEN Override := X2; END_IF;
IF E3 AND ABS(x3) > ABS(Override) THEN Override := X3; END_IF;

(* revision history
hm		4.11.2007		rev 1.0
	original version

*)
END_FUNCTION

(* POU engineering/signal processing/scale_B2, ST *)
FUNCTION scale_B2 : REAL
VAR_INPUT
	in1: BYTE;
	in2: BYTE;
	K : REAL;
	O : REAL;
END_VAR
VAR_INPUT CONSTANT
	in1_min: REAL := 0;
	in1_max: REAL := 1000;
	in2_min: REAL := 0;
	in2_max: REAL := 1000;
END_VAR

(*
version 1.2	6. jan 2008
programmer 	hugo
tested by		tobias

	this functiob block can scale up to two inputs.
	the inputs have their min value at 0 and their max value at 255 while the min and max value can be either positive or negative.
	the inputs ramp between min and max values for the respective inputs to be between (0..255).
	the summed output is then scaled by an scale input K and a offset O can be added to the output.
	the min and max input configurations can be edited in the cfc editor by double clicking the symbol body.

*)
scale_B2 := 	((in1_max - in1_min)* in1 * 0.00392156862 + in1_min +
				(in2_max - in2_min)* in2 * 0.00392156862 + in2_min)
				* K + O;

(* code bofore rev 1.2
scale_B2 := 	((in1_max - in1_min)* in1 / 255 + in1_min +
				(in2_max - in2_min)* in2 / 255 + in2_min)
				* K + O;
*)

(* revision History
hm 19.1.2007	rev 1.1
	changed outputs to real to avoid overflow of integer
	added offset for better cascading of scale functions
	changed from FB to function

hm	6. jan 2008	rev 1.2
	improved performance
*)
END_FUNCTION

(* POU engineering/signal processing/scale_B4, ST *)
FUNCTION scale_B4 : REAL
VAR_INPUT
	in1: BYTE;
	in2: BYTE;
	in3: BYTE;
	in4: BYTE;
	K : REAL;
	O : REAL;
END_VAR
VAR_INPUT CONSTANT
	in1_min: REAL := 0;
	in1_max: REAL := 1000;
	in2_min: REAL := 0;
	in2_max: REAL := 1000;
	in3_min: REAL := 0;
	in3_max: REAL := 1000;
	in4_min: REAL := 0;
	in4_max: REAL := 1000;
END_VAR

(*
version 1.2	6. jan 2008
programmer 	hugo
tested by		tobias

	this functiob block can scale up to 4 inputs.
	the inputs have their min value at 0 and their max value at 255 while the min and max value can be either positive or negative.
	the inputs ramp between min and max values for the respective inputs to be between (0..255).
	the summed output is then scaled by an scale input K and a offset O can be added to the output.
	the min and max input configurations can be edited in the cfc editor by double clicking the symbol body.

*)
scale_B4 := 	((in1_max - in1_min)* in1 * 0.00392156862 + in1_min +
				(in2_max - in2_min)* in2 * 0.00392156862 + in2_min +
				(in3_max - in3_min)* in3 * 0.00392156862 + in3_min +
				(in4_max - in4_min)* in4 * 0.00392156862 + in4_min)
				* K + O;

(* revision History
hm 19.1.2007	rev 1.1
	changed outputs to real to avoid overflow of integer
	added offset for better cascading of scale functions
	changed from fb to function

hm	6. jan 2008	rev 1.2
	improved performance
*)
END_FUNCTION

(* POU engineering/signal processing/scale_B8, ST *)
FUNCTION scale_B8 : REAL
VAR_INPUT
	in1: BYTE;
	in2: BYTE;
	in3: BYTE;
	in4: BYTE;
	in5: BYTE;
	in6: BYTE;
	in7: BYTE;
	in8: BYTE;
	K : REAL;
	O : REAL;
END_VAR
VAR_INPUT CONSTANT
	in1_min: REAL := 0;
	in1_max: REAL := 1000;
	in2_min: REAL := 0;
	in2_max: REAL := 1000;
	in3_min: REAL := 0;
	in3_max: REAL := 1000;
	in4_min: REAL := 0;
	in4_max: REAL := 1000;
	in5_min: REAL := 0;
	in5_max: REAL := 1000;
	in6_min: REAL := 0;
	in6_max: REAL := 1000;
	in7_min: REAL := 0;
	in7_max: REAL := 1000;
	in8_min: REAL := 0;
	in8_max: REAL := 1000;
END_VAR

(*
version 1.2	6. jan 2008
programmer 	hugo
tested by		tobias

	this functiob block can scale up to 8 inputs.
	the inputs have their min value at 0 and their max value at 255 while the min and max value can be either positive or negative.
	the inputs ramp between min and max values for the respective inputs to be between (0..255).
	the summed output is then scaled by an scale input K and a offset O can be added to the output.
	the min and max input configurations can be edited in the cfc editor by double clicking the symbol body.

*)
scale_B8 := 	((in1_max - in1_min)* in1 * 0.00392156862 + in1_min +
				(in2_max - in2_min)* in2 * 0.00392156862 + in2_min +
				(in3_max - in3_min)* in3 * 0.00392156862 + in3_min +
				(in4_max - in4_min)* in4 * 0.00392156862 + in4_min +
				(in5_max - in5_min)* in5 * 0.00392156862 + in5_min +
				(in6_max - in6_min)* in6 * 0.00392156862 + in6_min +
				(in7_max - in7_min)* in7 * 0.00392156862 + in7_min +
				(in8_max - in8_min)* in8 * 0.00392156862 + in8_min)
				* K + O;

(* revision History
hm 19.1.2007	rev 1.1
	changed outputs to real to avoid overflow of integer
	added offset for better cascading of scale functions

hm	6. jan 2008	rev 1.2
	improved performance
*)
END_FUNCTION

(* POU engineering/signal processing/scale_X2, ST *)
FUNCTION scale_X2 : REAL
VAR_INPUT
	in1: BOOL;
	in2: BOOL;
	K : REAL;
	O : REAL;
END_VAR
VAR_INPUT CONSTANT
	in1_min: REAL := 0;
	in1_max: REAL := 1000;
	in2_min: REAL := 0;
	in2_max: REAL := 1000;
END_VAR

(*
version 1.0	19 jan 2007
programmer 	hugo
tested by		tobias

	this functiob block can scale up to two inputs.
	the input can select between two values with true or false.
	the summed output is then scaled by an scale input K and a offset O can be added to the output.
	the min and max input configurations can be edited in the cfc editor by double clicking the symbol body.

*)
IF NOT in1 THEN scale_x2 := in1_min; ELSE scale_x2 := in1_max; END_IF;
IF NOT in2 THEN scale_x2 := scale_x2 + in2_min; ELSE scale_x2 := scale_x2 + in2_max; END_IF;
scale_X2 := scale_X2 * k + O;

(* revision history

*)
END_FUNCTION

(* POU engineering/signal processing/scale_X4, ST *)
FUNCTION scale_X4 : REAL
VAR_INPUT
	in1: BOOL;
	in2: BOOL;
	in3: BOOL;
	in4: BOOL;
	K : REAL;
	O : REAL;
END_VAR
VAR_INPUT CONSTANT
	in1_min: REAL := 0;
	in1_max: REAL := 1000;
	in2_min: REAL := 0;
	in2_max: REAL := 1000;
	in3_min: REAL := 0;
	in3_max: REAL := 1000;
	in4_min: REAL := 0;
	in4_max: REAL := 1000;
END_VAR

(*
version 1.0	19 jan 2007
programmer 	hugo
tested by		tobias

	this function can scale up to 4 inputs.
	the input can select between two values with true or false.
	the summed output is then scaled by an scale input K and a offset O can be added to the output.
	the min and max input configurations can be edited in the cfc editor by double clicking the symbol body.

*)
IF NOT in1 THEN scale_X4 := in1_min; ELSE scale_X4 := in1_max; END_IF;
IF NOT in2 THEN scale_x4 := scale_x4 + in2_min; ELSE scale_x4 := scale_x4 + in2_max; END_IF;
IF NOT in3 THEN scale_x4 := scale_x4 + in3_min; ELSE scale_x4 := scale_x4 + in3_max; END_IF;
IF NOT in4 THEN scale_x4 := scale_x4 + in4_min; ELSE scale_x4 := scale_x4 + in4_max; END_IF;
scale_X4 := scale_X4 * k + O;

(* revision history

*)
END_FUNCTION

(* POU engineering/signal processing/scale_X8, ST *)
FUNCTION scale_X8 : REAL
VAR_INPUT
	in1: BOOL;
	in2: BOOL;
	in3: BOOL;
	in4: BOOL;
	in5: BOOL;
	in6: BOOL;
	in7: BOOL;
	in8: BOOL;
	K : REAL;
	O : REAL;
END_VAR
VAR_INPUT CONSTANT
	in1_min: REAL := 0;
	in1_max: REAL := 1000;
	in2_min: REAL := 0;
	in2_max: REAL := 1000;
	in3_min: REAL := 0;
	in3_max: REAL := 1000;
	in4_min: REAL := 0;
	in4_max: REAL := 1000;
	in5_min: REAL := 0;
	in5_max: REAL := 1000;
	in6_min: REAL := 0;
	in6_max: REAL := 1000;
	in7_min: REAL := 0;
	in7_max: REAL := 1000;
	in8_min: REAL := 0;
	in8_max: REAL := 1000;
END_VAR

(*
version 1.0	19 jan 2007
programmer 	hugo
tested by		tobias

	this function can scale up to 4 inputs.
	the input can select between two values with true or false.
	the summed output is then scaled by an scale input K and a offset O can be added to the output.
	the min and max input configurations can be edited in the cfc editor by double clicking the symbol body.

*)
IF NOT in1 THEN scale_x8 := in1_min; ELSE scale_x8 := in1_max; END_IF;
IF NOT in2 THEN scale_x8 := scale_x8 + in2_min; ELSE scale_x8 := scale_x8 + in2_max; END_IF;
IF NOT in3 THEN scale_x8 := scale_x8 + in3_min; ELSE scale_x8 := scale_x8 + in3_max; END_IF;
IF NOT in4 THEN scale_x8 := scale_x8 + in4_min; ELSE scale_x8 := scale_x8 + in4_max; END_IF;
IF NOT in5 THEN scale_x8 := scale_x8 + in5_min; ELSE scale_x8 := scale_x8 + in5_max; END_IF;
IF NOT in6 THEN scale_x8 := scale_x8 + in6_min; ELSE scale_x8 := scale_x8 + in6_max; END_IF;
IF NOT in7 THEN scale_x8 := scale_x8 + in7_min; ELSE scale_x8 := scale_x8 + in7_max; END_IF;
IF NOT in8 THEN scale_x8 := scale_x8 + in8_min; ELSE scale_x8 := scale_x8 + in8_max; END_IF;
scale_X8 := scale_X8 * k + O;

(* revision history

*)
END_FUNCTION

(* POU Logic/gate logic/mux_2, ST *)
FUNCTION mux_2 : BOOL
VAR_INPUT
	D0: BOOL;
	D1: BOOL;
	A0: BOOL;
END_VAR
VAR
END_VAR

(*
	version 1.1	5 oct 2006
	programmer 	hugo
	tested BY		tobias

	dual input multiplexer
	depending on the value of A0, D0 or D1 will be switched to the Output

	executioin TIME on wago 750-841 = 7us
*)
mux_2 := (D0 AND NOT A0) OR (D1 AND A0);

(*

change history:
5.10.2006		rev 1.1
	changed to ST Langage for better protability.

*)
END_FUNCTION

(* POU Logic/gate logic/mux_4, ST *)
FUNCTION mux_4 : BOOL
VAR_INPUT
	D0: BOOL;
	D1: BOOL;
	D2: BOOL;
	D3: BOOL;
	A0: BOOL;
	A1: BOOL;
END_VAR
VAR
END_VAR

(*
	version 1.1	5 oct 2006
	programmer 	hugo
	tested BY		tobias

	quad input multiplexer
	depending on the value of A0 and A1, one of the 4 inputs will be switched to the Output

	executioin TIME on wago 750-841 = 13us
*)
mux_4 := (D0 AND NOT A0 AND NOT A1)
	OR (D1 AND A0 AND NOT A1)
	OR (D2 AND NOT A0 AND A1)
	OR (D3 AND A0 AND A1);


(* change history:

5.10.2006		rewritten to ST for better portability


*)
END_FUNCTION

(* POU Logic/gate logic/parity, ST *)
FUNCTION parity : BOOL
VAR_INPUT
	in : DWORD;
END_VAR
VAR
END_VAR

(*
	version 1.3	18 feb 2008
	programmer 	hugo
	tested BY		hans

this function calculates the even parity of an input Dword
the output will be true if the amount of high bits are an odd number.

*)
WHILE in > 0 DO
	parity := parity XOR in.0 XOR in.1 XOR in.2 XOR in.3;
	in := SHR(in,4);
END_WHILE;

(* code before rev 1.2
WHILE in > 0 DO
	IF in.0 THEN cnt := cnt +1; END_IF;
	in := SHR(in,1);
END_WHILE;
IF (cnt MOD 2) = 1 THEN parity := TRUE; ELSE parity := FALSE; END_IF;
*)

(* revision history

rev 1.0 hm 1 sep 2006
	original version

rev 1.1 hm 10.9.2007
	changed algorithm to improve performance

rev 1.2	hm	8 dec 2007
	changed algorithm to improve performance

rev 1.3	hm	18 feb 2008
	changed algorithm to improve performance
*)
END_FUNCTION

(* POU Logic/gate logic/SHL1, ST *)
FUNCTION SHL1 : DWORD
VAR_INPUT
	IN : DWORD;
	N : INT;
END_VAR
VAR CONSTANT
	temp : DWORD := 16#FFFF_FFFF;
END_VAR

(*
version 1.1	27 dec 2007
programmer 	hugo
tested by		tobias

SHL1 shifts N bits to the left filling the new bits with 1

*)
SHL1 := SHR(temp,32-N) OR SHL(IN,N);


(* revision history
hm	14.9.2007		rev 1.0
	original version

hm	27. dec 2007	rev 1.1
	changed code for better performance

*)
END_FUNCTION

(* POU Logic/gate logic/SHR1, ST *)
FUNCTION SHR1 : DWORD
VAR_INPUT
	IN : DWORD;
	N : INT;
END_VAR
VAR CONSTANT
	temp : DWORD := 16#FFFF_FFFF;
END_VAR

(*
version 1.1	27 dec 2007
programmer 	hugo
tested by		tobias

SHR1 shifts N bits to the right filling the new bits with 1

*)
SHR1 := SHL(temp,32-N) OR SHR(IN,N);

(* revision history
hm	14.9.2007		rev 1.0
	original version

hm	27. dec 2007	rev 1.1
	changed code for better performance

*)
END_FUNCTION

(* POU Logic/gate logic/Word_of_Byte, ST *)
FUNCTION Word_of_Byte : WORD
VAR_INPUT
	B0 : BYTE;
	B1 : BYTE;
END_VAR
VAR
END_VAR

(*
version 1.2	19. feb 2008
programmer 	hugo
tested by		tobias

this function creates a word from 2 individual bytes

*)
Word_of_Byte := SHL(B1,8) OR B0;

(* revision history
hm	24. jan 2007	rev 1.0
	original version

hm	2. jan 2008		rev 1.1
	improved performance

hm	19. feb 2008	rev 1.2
	replaced and with or for better compatibility

*)
END_FUNCTION

(* POU Logic/gate logic/Word_of_Dword, ST *)
FUNCTION Word_of_Dword : WORD
VAR_INPUT
	in : DWORD;
	N : BYTE;
END_VAR
VAR
END_VAR

(*
version 1.1	2 jan 2008
programmer 	hugo
tested by		tobias

this function extracts a single word from the nth position from right (right is lowest byte)
the lower word (starting weith Bit0 from in) is selected with N=0.
*)
Word_of_Dword := DWORD_TO_WORD(SHR(in,n*16));

(* revision history
hm	17. jan 2007	rev 1.0
	original version

hm	2. jan 2008		rev 1.1
	improved performance

*)
END_FUNCTION

(* POU mathematical/Geometry/sphere_V, ST *)
FUNCTION sphere_V : REAL
VAR_INPUT
	rx : REAL;
END_VAR
VAR
END_VAR

(*
version 1.2	22. feb 2008
programmer 	hugo
tested by		tobias

sphere_V calculates the Volume of a Sphere


*)
sphere_V := 4.188790205 * Rx * RX * RX;

(* revision histroy
hm	16. oct 2007	rev 1.0
	original version

hm	4. dec 2007		rev 1.1
	changed code for better performance

hm	22. feb 2008		rev 1.2
	changed code for better performance
*)
END_FUNCTION

(* POU mathematical/Geometry/triangle_A, ST *)
FUNCTION triangle_A : REAL
VAR_INPUT
	S1 : REAL;
	A : REAL;
	S2 : REAL;
	S3 : REAL;
END_VAR
VAR
END_VAR

(*
version 1.1	22. feb 2008
programmer 	hugo
tested by		tobias

triangle_A calculates the Area of a triangle.
if any input is 0 it will be neglected and the are will be calculated from eiter:
two sides and an angle (s1 and S2 and the angle A1) or 3 sides.


*)
IF A = 0 THEN
	triangle_A := SQRT((s1+s2+S3) * (s1+s2-S3) * (S2+S3-S1) * (S3+S1-S2)) * 0.25;
ELSE
	triangle_A := S1 * S2 * SIN(Rad(A)) * 0.5;
END_IF;

(* revision histroy
hm	16. oct 2007	rev 1.0
	original version

hm	22. feb 2008	rev 1.1
	improved performance
*)
END_FUNCTION

(* POU mathematical/Vektormathematik/V3_NUL, ST *)
FUNCTION V3_NUL : BOOL
VAR_INPUT
	A : Vector_3;
END_VAR
VAR
END_VAR

(*
version 1.0	12 dec 2007
programmer 	hugo
tested by		tobias

this function checks if a vectors in a null Vector

*)
V3_NUL := A.X = 0 AND A.Y = 0 AND A.Z = 0;



(* revision history
hm		12 dec 2007	rev 1.0
	original version

*)
END_FUNCTION

(* POU mathematical/gamma, ST *)
FUNCTION gamma : REAL
VAR_INPUT
	X : REAL;
END_VAR
VAR
END_VAR

(*
version 1.0	10 dec 2007
programmer 	hugo
tested by		tobias

this function calculates the stirling function which is an approximation for the gamma function

*)
IF X >=0 THEN gamma := SQRT(pi2*X)*EXPT(X/E,X); END_IF;

(* revision history
hm	10.12.2007	rev 1.0
	original version

*)
END_FUNCTION

(* POU mathematical/max3, ST *)
FUNCTION max3 : REAL
VAR_INPUT
	in1 : REAL;
	in2 : REAL;
	in3 : REAL;
END_VAR
VAR
END_VAR

(*
version 1.0	1 jan 2007
programmer 	hugo
tested by		tobias

this function returns the highest of 3 real values

*)
IF in1 >= in2 AND in1 >= in3 THEN
	max3 := in1;
ELSIF in2 >= in1 AND in2 >= in3 THEN
	max3 := in2;
ELSE
	max3 := in3;
END_IF;
END_FUNCTION

(* POU mathematical/min3, ST *)
FUNCTION min3 : REAL
VAR_INPUT
	in1 : REAL;
	in2 : REAL;
	in3 : REAL;
END_VAR
VAR
END_VAR

(*
version 1.0	1 jan 2007
programmer 	hugo
tested by		tobias

this function returns the lowest of 3 real values

*)
IF in1 <= in2 AND in1 <= in3 THEN
	min3 := in1;
ELSIF in2 <= in1 AND in2 <= in3 THEN
	min3 := in2;
ELSE
	min3 := in3;
END_IF;
END_FUNCTION

(* POU mathematical/MUL_ADD, ST *)
FUNCTION MUL_ADD : REAL
VAR_INPUT
	X : REAL;
	K : REAL;
	O : REAL;
END_VAR
VAR
END_VAR

(*
version 1.1	11 nov 2007
programmer 	hugo
tested by		tobias

this function multiplies an input X with K and adds Offset O to the result.

*)
MUL_ADD := X * K + O;

(* revision history
hm	28. feb 2007
	original version

hm	11.nov 2007		rev 1.1
	deleted preset values for K and O this makes no sense for a function

*)
END_FUNCTION

(* POU mathematical/round, ST *)
FUNCTION round : REAL
VAR_INPUT
	in : REAL;
	N : INT;
END_VAR
VAR
	X: REAL;
END_VAR

(*
version 1.2	8. jan 2008
programmer 	hugo
tested by	tobias

this function rounds a real down to n digits behind the comma.
round(3.1415,1) = 3.1

*)
IF N < 4 THEN
	IF N < 2 THEN
		IF N = 0 THEN X := 1; ELSE X := 10; END_IF;
	ELSE
		IF N = 2 THEN X := 100; ELSE X := 1000; END_IF;
	END_IF;
ELSE
	IF N < 6 THEN
		IF N = 4 THEN X := 10000; ELSE X := 100000; END_IF;
	ELSE
		IF N = 6 THEN X := 1000000; ELSE X := 10000000; END_IF;
	END_IF;
END_IF;

round := TRUNC(in * X + 0.5) / X;

(* revision history
hm	1. sep 2006	rev 1.0
	original version

hm	2. dec 2007	rev 1.1
	changed code for better performance

hm	8. jan 2008	rev 1.2
	further improvement in performance
*)
END_FUNCTION

(* POU mathematical/sign_I, ST *)
FUNCTION sign_I : BOOL
VAR_INPUT
	in : INT;
END_VAR
VAR
END_VAR

(*
version 1.2	1 dec 2007
programmer 	hugo
tested by	tobias

this function return true if the integer input is negative

*)
sign_I := in.15;

(* revision history
hm 3.3.2007	rev 1.1
	changed method of function for better compatibility to other systems

hm	1.12.2007	rev 1.2
	changed code to improve performance
*)
END_FUNCTION

(* POU mathematical/sqrtn, ST *)
FUNCTION sqrtn : REAL
VAR_INPUT
	X : REAL;
	N : INT;
END_VAR
VAR
END_VAR

(*
version 1.1	2 dec 2007
programmer 	hugo
tested by	tobias

this function calculates the nth root function of X according to the formula sqrtn = x^(1/n).

*)
IF N > 0 THEN
(*	sqrtn := EXPT(x, 1.0 / INT_TO_REAL(n)); old code in rev 1.0 *)
sqrtn := EXP(LN(x)/n);
END_IF;

(* revision history
hm		12 jan 2007	rev 1.0
	original version

hm		2. dec 2007	rev 1.1
	changed code for better performance

*)
END_FUNCTION

(* POU mathematical/tanH, ST *)
FUNCTION tanH : REAL
VAR_INPUT
	X : REAL;
END_VAR
VAR
END_VAR


(*
version 1.1	1 dec 2007
programmer 	hugo
tested by	tobias

this function calculates the tangens hyperbolicus

*)
tanH := -2 / (EXP(-2 * x) + 1) + 1;

(* revision hisdtory
hm	12.1.2007	rev 1.0
	original version
hm	1.12.2007	rev 1.1
	changed code to improve performance
*)
END_FUNCTION

(* POU mathematical/window, ST *)
FUNCTION window : BOOL
VAR_INPUT
	low : REAL;
	in : REAL;
	high : REAL;
END_VAR
VAR
END_VAR

(*
	version 1.1	22 jan 2007
	programmer 	hugo
	tested BY	tobias

this checks a signal if the signal is between the upper and lower limit
*)
window := in < high AND in > low;


(* revision history
hm	22.1.2007	rev 1.1
	changed the order of inputs to low, in, high

*)
END_FUNCTION

(* POU mathematical/window2, ST *)
FUNCTION window2 : BOOL
VAR_INPUT
	low : REAL;
	in : REAL;
	high : REAL;
END_VAR
VAR
END_VAR

(*
	version 1.0	31 oct 2007
	programmer 	hugo
	tested BY	tobias

this checks a signal if the signal is between the upper and lower limit including the two limits
*)
window2 := in <= high AND in >= low;


(* revision history
hm	31.10.2007	rev 1.0
	original version

*)
END_FUNCTION

(* POU String/find_nonum, ST *)
FUNCTION find_nonum : INT
VAR_INPUT
	str : STRING;
END_VAR
VAR
	pos: INT;
	pt : POINTER TO BYTE;
END_VAR

(*
version 1.0	6 oct 2006
programmer 	hugo
tested by		tobias

find_noNum searches str and returns the first position which is not a number.
a number is characterized by a letter "0..9" or "."

*)
pt := ADR(str);
find_nonum := 0;
FOR pos := 1 TO LEN(str) DO;
	IF NOT((PT^ > 47 AND PT^ < 58) OR PT^ = 46) THEN
		find_nonum := pos;
		RETURN;
	END_IF;
	PT := PT + 1;
END_FOR;
END_FUNCTION

(* POU String/find_Num, ST *)
FUNCTION find_Num : INT
VAR_INPUT
	str : STRING;
END_VAR
VAR
	pos: INT;
	pt : POINTER TO BYTE;
END_VAR

(*
version 1.0	6 oct 2006
programmer 	hugo
tested by		tobias

find_Num searches str and returns the starting position of a number
a number is characterized by a letter "0..9" or "."

*)
pt := ADR(str);
find_Num := 0;
FOR pos := 1 TO LEN(str) DO;
	IF (PT^ > 47 AND PT^ < 58) OR PT^ = 46 THEN
		find_Num := pos;
		RETURN;
	END_IF;
	PT := PT + 1;
END_FOR;
END_FUNCTION

(* POU String/FindB, ST *)
FUNCTION FindB : INT
VAR_INPUT
	str1 : STRING;
	str2 : STRING;
END_VAR
VAR
	pos: INT;
	length: INT;
END_VAR

(*
version 1.1	15 dec 2007
programmer 	hugo
tested by		tobias

the function find searches an str1 for the presence of str2 and returns the first position of str1 of the last presence in instring.
the function is similar to find except it searches from the right to left.
 a 0 is returned if the string is not found.

*)
length := LEN(str2);
FOR pos := LEN(str1) - length + 1 TO 1 BY -1 DO
	IF MID(str1,length,pos) = str2 THEN
		FindB := pos;
		RETURN;
	END_IF;
END_FOR;

(* revision history
hm		6. oct 2006	rev 1.0
	original version

hm		15 dec 2007	rev 1.1
	changed code for better performance

*)
END_FUNCTION

(* POU String/HEX_TO_DWORD, ST *)
FUNCTION HEX_TO_DWORD : DWORD
VAR_INPUT
	Hex : STRING;
END_VAR
VAR
	pt : POINTER TO BYTE;
	i: INT;
	X: BYTE;
END_VAR

(*
version 1.1	19 nov 2007
programmer 	hugo
tested by		tobias

HEX_TO_DWORD converts a Hexadecimal string into a DWORD.

*)
pt := ADR(hex);
FOR I := 1 TO LEN(hex) DO
	(* read the first character and subtract 48 to get value in decimal 0 = 48 *)
	x := pt^ - 48;
	(* subtract again 7 IF value is higher THEN 9 A = 65 *)
	IF X > 9 THEN X := X - 7; END_IF;
	(* add up the output per hex character which is 4 bits wide *)
	HEX_TO_DWORD := SHL(HEX_TO_DWORD,4) + X;
	pt := pt + 1;
END_FOR

(* revision histroy
hm		2.10.2007		rev 1.0
	original release

hm		19.11.2007	rev 1.1
	changed type of function from int to dword

*)	
END_FUNCTION

(* POU String/lowercase, ST *)
FUNCTION lowercase : STRING
VAR_INPUT
	str : STRING;
END_VAR
VAR
	PT : POINTER TO BYTE;
	pos: INT;
	l: INT;
END_VAR

(*
version 1.1	4. feb 2008
programmer 	hugo
tested by		tobias

uppercase returns str while all letters A..Z and Ä.Ö,Ü are converted to lowercase.

*)
PT := ADR(lowercase);
lowercase := str;
l := LEN(str);
FOR pos := 1 TO l DO
	IF (PT^ > 64 AND PT^ < 91) OR pt^ = 196 OR pt^ = 214 OR pt^ = 220 THEN PT^ := PT^ + 32; END_IF;
	PT := PT + 1;
END_FOR;

(* revision histroy
hm		6.10.2006		rev 1.0
	original release

hm		4.2.2008		rev 1.1
	improved performance
	added Ä.Ö,Ü
*)	
END_FUNCTION

(* POU String/Real_To_StrF, ST *)
FUNCTION Real_To_StrF : STRING
VAR_INPUT
	IN : REAL;
	N : INT;
END_VAR
VAR
	temp : DWORD := 1;
	I: INT;
	L: INT;
	p1, p2 : POINTER TO BYTE;
END_VAR

(*
version 1.2	15 dec 2007
programmer 	hugo
tested by		tobias

Real_to_strF converts a Real to a fixed length String.
the string will be filles with leading zeroes to achieve the fixed length after the dot, or if too long, the lowest digits will be discarded.


*)
(* read pointer to output *)
p1 := ADR(Real_To_StrF);
p2 := p1;

(* multiply in with 10^N and truncate *)
FOR I := 1 TO N DO
	temp := temp * 10;
END_FOR;
(* multiply temp with in to shift n digits to the left *)
temp := TRUNC(in * temp);
Real_To_StrF := DWORD_TO_STRING(temp);
(* now take care of the dot at length - Nth position *)
L := LEN(Real_To_StrF);
(* we need to add zero's at the end of the string if there are less then N + 1 zeroes *)
(* this for loop is to align the pointer p1 to the end of the string *)
FOR i := 1 TO L DO p1 := p1 + 1; END_FOR;
FOR i := L TO N DO
	p1^ := 48;
	p1 := p1 + 1;
END_FOR;
(* now we create the space for the dot *)
p2 := p1 - 1;
FOR i := 1 TO N DO
	p1^ := p2^;
	p1 := p1 - 1;
	p2 := p2 - 1;
END_FOR;
(* now we add the dot if N > 0 *)
IF N > 0 THEN
	p1^ := 46;
	(* the string needs to be closed with a 0 at the end *)
	FOR i := 1 TO N + 1 DO p1 := p1 + 1; END_FOR;
	p1^ := 0;
END_IF;


(* code before rev 1.2
dw1 := TRUNC(ABS(in));
dw2 := TRUNC(fract(ABS(in))*exp10(N)+0.5);
IF in < 0 THEN
	s1 := CONCAT('-', DWORD_TO_STRING(dw1));
ELSE
	s1 := DWORD_TO_STRING(dw1);
END_IF;
IF N > 0 THEN s1 := CONCAT(s1, '.'); END_IF;
s2 := DWORD_To_STRF(dw2,N);
Real_To_StrF := CONCAT(s1, s2);
*)

(* revision history
hm		26 jan 2007	rev 1.0
	original version

hm		20. nov 2007	rev 1.1
	when N=0 ther will be no dot at the end of the string.

hm		15 dec 2007		rev 1.2
	changed code for better performance

*)
END_FUNCTION

(* POU Time&Date/hour_to_time, ST *)
FUNCTION hour_to_time : TIME
VAR_INPUT
	input : REAL;
END_VAR
VAR
END_VAR

(*
version 1.0	4 aug 2006
programmer 	hugo
tested by		tobias

converts an amount of hours in real to time

*)
hour_to_time := DWORD_TO_TIME(REAL_TO_DWORD(input * 3600000));
END_FUNCTION

(* POU Time&Date/leap_year, ST *)
FUNCTION leap_year : BOOL
VAR_INPUT
	yr : INT;
END_VAR
VAR
END_VAR

(*
version 1.1	2 oct 2006
programmer 	hugo
tested by		tobias


leap_year is true if the tested year is a leap year  
execution time on wago 750-841 =  12 us    
*)
leap_year := SHL(yr,14) = 0;

(* this code was used prior to rev 1.1

IF yr MOD 400 = 0 THEN leap_year := TRUE;
ELSIF yr MOD 100 = 0 THEN leap_year := FALSE;
ELSIF yr MOD 4 =0 THEN leap_year := TRUE;
ELSE leap_year := FALSE;
END_IF;

*)

(* change history

hm 	2.10.2006		rev 1.1
	the function now works for any year from 1970 up to 2100

hm	1. oct 2007		rev 1.2
	chaged code for higher performance
*)
END_FUNCTION

(* POU Time&Date/local_time, ST *)
FUNCTION local_time : DT
VAR_INPUT
	utc : DT;
	time_zone_offset : INT;
	dst_enable: BOOL;
END_VAR
VAR
	tx : TIME;
END_VAR

(*
version 1.4	8 dec 2007
programmer 	hugo
tested by		tobias

localtime calculates the local time according to DSTenable and time_zone_offset.
the dst input only tells the function the dst (daylight savings time) is enabled but the calculation for summertime on and off is done by the function itself.
this means the dst input only tells the function to switch summertime on and off automatically or not.
the function will switch to summertime automatically at the specified time end of march and back end of october.
the summertime calculation is done according to european standards.
the input is world time (UTC) and a given time_zone_offset for any time_zone.

execution time on wago 750-841 = 140 us   
*)
tx := DWORD_TO_TIME(INT_TO_DWORD(ABS(time_zone_offset))* 3600000);

IF DST(utc) AND dst_enable THEN
	IF time_zone_offset < 0 THEN local_time := utc - tx + T#1h; ELSE local_time := utc + tx + T#1h; END_IF;
ELSE
	IF time_zone_offset < 0 THEN local_time := utc - tx; ELSE local_time := utc + tx; END_IF;
END_IF;


(*

change history

2.10.2006 hm	rev 1.1
	corrected an error in the dst check for correct function

24. oct 2007	rev 1.2
	changed dst calculation because function dst was upgraded no error in DCF77 only a change in DST

12. nov 2007	rev 1.3
	changed time_zone_offset from time to integer to allow for negative offset time zones

8 dec 2007		rev 1.4
	corrected a problem with time_zone_offset
*)
END_FUNCTION

(* POU Time&Date/Ltime_to_UTC, ST *)
FUNCTION Ltime_to_UTC : DT
VAR_INPUT
	Ltime : DT;
	DST : BOOL;
	Time_Zone_Offset : INT;
END_VAR
VAR
	dst_offset : TIME := T#1h;
	tx: TIME;
END_VAR

(*
version 1.3		8 dec 2007
programmer 	hugo
tested by		tobias

LTIME_TO_UTC calculates UTC (World Time) from a local time LTIME. utc is calculated by subtracting Time_Zone_Offset from ltime and if dst it true subtracting an additional hour from ltime.

*)
(* convert integer time_zone_offset to hours *)
tx := DWORD_TO_TIME(INT_TO_DWORD(ABS(time_zone_offset))* 3600000);

IF DST THEN
	IF time_zone_offset < 0 THEN
		Ltime_to_UTC := Ltime + tx - dst_offset;
	ELSE
		Ltime_to_UTC := Ltime - tx - dst_offset;
	END_IF;
ELSE
	IF time_zone_offset < 0 THEN
		Ltime_to_UTC := Ltime + tx;
	ELSE
		Ltime_to_UTC := Ltime - tx;
	END_IF;
END_IF;



(* revision history
hm 5.7.2007		rev 1.0		
	original version

hm 5.11.2007	rev 1.1
	replaced literal constant with variable because of error in möller ecp4 compiler

hm	12.nov 2007	rev 1.2
	changed Type of time_zone_offset from time to int to allow for time zones with negative offset

hm	8. dec 2007	rev 1.3
	corrected a problem with time_zone_offset
*)
END_FUNCTION

(* POU Time&Date/minute_to_time, ST *)
FUNCTION minute_to_time : TIME
VAR_INPUT
	input : REAL;
END_VAR
VAR
END_VAR

(*
version 1.0	4 aug 2006
programmer 	hugo
tested by		tobias

converts an amount of minutes in real to time
execution time on wago 750-841 =  17us
*) 
minute_to_time := DWORD_TO_TIME(REAL_TO_DWORD(input * 60000));
END_FUNCTION

(* POU Time&Date/period, ST *)
FUNCTION period : BOOL
VAR_INPUT
	d1 : DATE;
	dx : DATE;
	d2 : DATE;
END_VAR
VAR
	day1, day2, dayx : INT;
END_VAR

(*
version 1.2	4 jan 2008
programmer 	hugo
tested by		tobias

PERIOD checks if a given date is between two dates (d1 and d2) d1 is the starting date and d2 the last date for the period.
the years of the dates are ignored, so the function period cheks for a time period within a year independet of the year.

*)
day1 := day_of_year(d1);
day2 := day_of_year(d2);
dayx := day_of_year(dx);
IF leap_of_Date(dx) AND dayx > 59 THEN dayx := dayx - 1; END_IF;

IF day2 < day1 THEN
	(* the period spans over the new year *)
	period := dayx <= day2 OR dayx >= day1;
ELSE
	period := dayx >= day1 AND dayx <= day2;
END_IF;

(* code before rev 1.2
yx := year(dx);
p1 := date_add(d1,0,0,0,yx - year(d1));
p2 := date_add(d2,0,0,0,yx - year(d2));

IF p2 >= p1 THEN
	period := dx <= p2  AND dx >= p1;
ELSE
	period := dx <= p2 OR dx >= p1;
END_IF;
*)


(* revision history

hm		19. sep 2007		rev 1.0
	original version

hm		20. sep 2007		rev 1.1
	corrected a problem with leap year

hm		4. jan 2008		rev 1.2
	changed code for better performance
*)
END_FUNCTION

(* POU Time&Date/second_to_time, ST *)
FUNCTION second_to_time : TIME
VAR_INPUT
	input : REAL;
END_VAR
VAR
END_VAR

(*
version 1.0	4 aug 2006
programmer 	hugo
tested by		tobias

converts an amount of seconds in real to time
execution TIME on wago 750-841 =  17us 

*)
second_to_time := DWORD_TO_TIME(REAL_TO_DWORD(input * 1000));
END_FUNCTION

(* POU Time&Date/set_Tod, ST *)
FUNCTION set_Tod : TOD
VAR_INPUT
	hour : INT;
	minute : INT;
	second : REAL;
END_VAR
VAR
END_VAR

(*
version 1.3	2 nov 2007
programmer 	hugo
tested by		tobias

creates tod from hour minute and second 

*)
set_Tod := DWORD_TO_TOD(DINT_TO_DWORD(TRUNC(second * 1000) + INT_TO_DINT(minute) * 60000 + INT_TO_DINT(hour) * 3600000));

(* revision history

hm		4.aug.2006		rev 1.0
	original version

hm		11. sep 2007	rev 1.1
	changed coding to avoid a compiler warning under twincat.

hm		1. nov 2007		rev 1.2
	changed coding to avoid possible overrun situation on möller ecp4

hm		2. Nov	2007	rev 1.3
	changed dword to DINT in calcualtion to avoid warnings with some compilers
*)
END_FUNCTION

(* POU Time&Date/work_week, ST *)
FUNCTION work_week : INT
VAR_INPUT
	idate : DATE;
END_VAR
VAR
	d1 : DATE;
	w1 : INT;
	ds: DWORD;
	yr: INT;
	w31: INT;
	w01: INT;
	wm: INT;
END_VAR

(*
version 1.2	19 dec 2007
programmer 	hugo
tested by		tobias

calculates the work week for a given date according to iso8601

*)
(* berechne den 1.1 des jahres von idate. *)
yr := year(idate);
d1 := year_begin(yr);
(* wochentag von d1 *)
w1 := weekday(d1);
(* offset des montags der eletzten KW des vorjahres *)
(* wenn der erste tag des jahres größer als donnerstag ist dann beginnt die letzte kw am montag davor *)
(* wenn der erste tag des jahres ein donnerstag oder kleiner ist beginnt die erste kw 2 montage davor *)
IF w1 < 5 THEN
	ds := DATE_TO_DWORD(d1) - (w1+6) * 86400;
ELSE
	ds := DATE_TO_DWORD(d1) + (1-w1) * 86400;
END_IF;

(* kalenderwoche des eingangsdatums *)
work_week := DWORD_TO_INT((DATE_TO_DWORD(idate) - ds) / 604800);

(* korrektur wenn work_week = 0 *)
IF work_week = 0 THEN
	(* work_week needs to be 53 when 1.jan of the year before is thursday or dec 31. is thursday. *)
	(* first and last weekday of a year is equal and one more day for a leap_year. *)
	IF w1 > 1 THEN w31 := w1 - 1; ELSE W31 := 7; END_IF;
	IF leap_year(yr - 1) THEN IF w31 > 1 THEN w01 := W31 - 1; ELSE w1 := 7; END_IF; END_IF;
	(* if first or last day of a year is a thursday, the year has 53 weeks *)
	IF w31 = 4 OR w01 = 4 THEN work_week := 53; ELSE work_week := 52; END_IF;
ELSE
	(* end of year calculation *)
	(* calculated the first and last weekday *)
	IF leap_year(yr) THEN
		IF w1 < 7 THEN w31 := w1 + 1; ELSE w31 := 1; END_IF;
	ELSE
		w31 := w1;
	END_IF;
	(* if first or last day is thursday then the year has 53 weeks otherwise only 52 *)
	IF w31 = 4 OR w1 = 4 THEN wm := 53; ELSE wm := 52; END_IF;
	IF work_week > wm THEN work_week := 1; END_IF;
END_IF;



(* old code before rev 1.2
w1 := weekday(set_Date(year(idate), 1,1));
IF w1 < 5 THEN
	work_week := (day_of_year(idate) + w1 + 5)/7;
ELSE
	work_week := (day_of_year(idate) + w1 - 2)/7;
END_IF
*)


(* revision history

hm 17.1.2007		rev 1.1
	deleted unused variable yday

hm	19. dec 2007	rev 1.2
	changed code for better performance
*)
END_FUNCTION

(* POU mathematical/fib, ST *)
FUNCTION fib : REAL
VAR_INPUT
	X : INT;
END_VAR
VAR
	t1, t2: REAL;
END_VAR

(*
version 1.1	2 jan 2008
programmer 	hugo
tested by		tobias

this function calculates the fibonacci sequence

*)
IF x < 2 THEN
	fib := X;
	RETURN;
ELSE
	(* the fibonacci number is the sum of the two suceeding fibonaci numbers *)
	(* we store the numbers alternatively in t1 and t2 depending on pt *)
	t2 := 1;
	WHILE X > 3 DO
		X := X-2;
		t1 := t1 + t2;
		t2 := t1 + t2;
	END_WHILE;
	IF X > 2 THEN t1 := t1 + t2; END_IF;
	fib := t1 + t2;
END_IF;

(* alternative code for very big numbers

IF X < 31 THEN
	fib := 0.4472136 * (expn(1.618034,X) - expn(-0.618034,X));
ELSE
	fib := 0.4472133 * expn(1.618034,X);
END_IF;

*)

(* revision history
hm	27. dec 2007	rev 1.0
	original version

hm	2. jan 2008		rev 1.1
	deleted unused variable pt
*)
END_FUNCTION

(* POU String/FINDP, ST *)
FUNCTION FINDP : INT
VAR_INPUT
	str : STRING;
	src : STRING;
	pos: INT;
END_VAR
VAR
	i: INT;
	ls: INT;
	lx: INT;
	stp: INT;
END_VAR

(*
version 1.0	4 feb 2008
programmer 	hugo
tested by		tobias

the function findP searches a string str for the occurence of src beginning at the position pos.

*)
ls := LEN(str);
lx := LEN(src);
IF ls < lx OR lx = 0 THEN RETURN; END_IF;
stp := ls - lx + 1;
FOR i := pos TO stp DO
	IF MID(str,lx,i) = src THEN
		FINDP := i;
		EXIT;
	END_IF;
END_FOR;

(* revision histroy
hm		4. feb. 2008		rev 1.0
	original release

*)	
END_FUNCTION

(* POU XTEST/Ideas/FM_INVSQRT, ST *)
FUNCTION FM_INVSQRT : REAL
VAR_INPUT
	X: REAL;
END_VAR
VAR
	PTR : POINTER TO DWORD;
	XHALF: REAL;
END_VAR
XHALF := X * 0.5;
ptr := ADR(X);
ptr^ := 16#5F375A86 - SHR(ptr^,1);
FM_INVSQRT := X * (1.5 - XHALF * X * X);
END_FUNCTION

(* POU XTEST/Ideas/I2C, ST *)
FUNCTION_BLOCK I2C
VAR_INPUT
	scl_in : BOOL;
	sda_in : BOOL;
END_VAR
VAR_OUTPUT
	scl_out : BOOL;
	sda_out : BOOL;
	busy: BOOL;
	error: BOOL;
END_VAR
VAR
	state : INT;
END_VAR
(* the following state machine is responsible for all actions on the I2C Bus *)
CASE state OF
	0:	(* no actions *)
		busy := FALSE;

	1: (* ready for transfer *)
		RETURN;

	10: (* generate start condition *)
		busy := TRUE;
		IF sda_in AND scl_in THEN
			(* bus is free, start sequence can be completed *)
			sda_out := FALSE;
			state := 11;
		ELSIF NOT scl_in AND sda_in THEN
			(* if scl is low and sda is true then scl needs to go high first *)
			scl_out := TRUE;
		ELSIF NOT scl_in AND NOT sda_in THEN
			(* both scl and sda are low sda need to go high first *)
			sda_out := TRUE;
		ELSIF NOT scl_in AND NOT sda_in THEN
			(* both scl and sda are low scl need to go low first *)
			scl_out := FALSE;
		END_IF;
	11: (* second phase of start cycle, pull scl low *)
		scl_out := FALSE;
		state := 1;

	20:	(* generate stop condition *)
		busy := TRUE;
		IF scl_in AND NOT sda_in THEN
			(* scl is high and sda is low sequence can be completed *)
			sda_out := TRUE;
			state := 0;
		ELSIF NOT scl_in AND NOT sda_in THEN
			(* scl and sda are low,  scl need to go high first *)
			scl_out := TRUE;
		ELSIF NOT scl_in AND sda_in THEN
			(* scl is low and sda is high, sda need to go low first *)
			sda_out := FALSE;
		ELSIF scl_in AND sda_in THEN
			(* scl and sda are high, scl need to go low first *)
			scl_out := FALSE;
		END_IF;

	30:	(* master acknowledge cycle *)
		IF NOT busy AND scl_in THEN
			(* if no transfer takes place an acknowledge cannot be received *)
			error := TRUE;
		ELSIF TRUE THEN
			(* bring sda true to check for ack *)
			sda_out := TRUE;
		END_IF;



END_CASE
END_FUNCTION_BLOCK

(* POU Device Drivers/IRTRANS_1, ST *)
FUNCTION_BLOCK IRTRANS_1
VAR_INPUT CONSTANT
	device_code : STRING;
	key_code : STRING;
END_VAR
VAR_INPUT
	cmd : BOOL;
END_VAR
VAR_IN_OUT
	device : STRING;
	key : STRING;
END_VAR
VAR_OUTPUT
	Q : BOOL;
END_VAR
VAR
END_VAR

(*
	version 1.0	2 jan 2008
	programmer 	hugo
	tested BY		tobias

*)
IF cmd AND device_code = device AND key_code = key THEN
	Q := TRUE;
ELSE
	Q := FALSE;
END_IF;

(* revision history
hm	2. jan 2008		rev 1.0
	original version

*)
END_FUNCTION_BLOCK

(* POU Device Drivers/IRTRANS_4, ST *)
FUNCTION_BLOCK IRTRANS_4
VAR_INPUT CONSTANT
	device_code : STRING;
	key_code_0 : STRING;
	key_code_1 : STRING;
	key_code_2 : STRING;
	key_code_3 : STRING;
END_VAR
VAR_INPUT
	cmd : BOOL;
END_VAR
VAR_IN_OUT
	device : STRING;
	key : STRING;
END_VAR
VAR_OUTPUT
	Q0, Q1, Q2, Q3 : BOOL;
END_VAR
VAR
END_VAR

(*
	version 1.0	2 jan 2008
	programmer 	hugo
	tested BY		tobias

*)
Q0 := FALSE;
Q1 := FALSE;
Q2 := FALSE;
Q3 := FALSE;
IF cmd AND device_code = device THEN
	IF key = key_code_0 THEN q0 := TRUE;
	ELSIF key = key_code_1 THEN q1 := TRUE;
	ELSIF key = key_code_2 THEN q2 := TRUE;
	ELSIF key = key_code_3 THEN q3 := TRUE;
	END_IF;
END_IF;

(* revision history
hm	2. jan 2008		rev 1.0
	original version

*)
END_FUNCTION_BLOCK

(* POU Device Drivers/IRTRANS_8, ST *)
FUNCTION_BLOCK IRTRANS_8
VAR_INPUT CONSTANT
	device_code : STRING;
	key_code_0 : STRING;
	key_code_1 : STRING;
	key_code_2 : STRING;
	key_code_3 : STRING;
	key_code_4 : STRING;
	key_code_5 : STRING;
	key_code_6 : STRING;
	key_code_7 : STRING;
END_VAR
VAR_INPUT
	cmd : BOOL;
END_VAR
VAR_IN_OUT
	device : STRING;
	key : STRING;
END_VAR
VAR_OUTPUT
	Q0, Q1, Q2, Q3, Q4, Q5, Q6, Q7 : BOOL;
END_VAR
VAR
END_VAR

(*
	version 1.0	2 jan 2008
	programmer 	hugo
	tested BY		tobias

*)
Q0 := FALSE;
Q1 := FALSE;
Q2 := FALSE;
Q3 := FALSE;
Q4 := FALSE;
Q5 := FALSE;
Q6 := FALSE;
Q7 := FALSE;
IF cmd AND device_code = device THEN
	IF key = key_code_0 THEN q0 := TRUE;
	ELSIF key = key_code_1 THEN q1 := TRUE;
	ELSIF key = key_code_2 THEN q2 := TRUE;
	ELSIF key = key_code_3 THEN q3 := TRUE;
	ELSIF key = key_code_4 THEN q4 := TRUE;
	ELSIF key = key_code_5 THEN q5 := TRUE;
	ELSIF key = key_code_6 THEN q6 := TRUE;
	ELSIF key = key_code_7 THEN q7 := TRUE;
	END_IF;
END_IF;

(* revision history
hm	2. jan 2008		rev 1.0
	original version

*)
END_FUNCTION_BLOCK

(* POU Device Drivers/IRTRANS_DECODE, ST *)
FUNCTION_BLOCK IRTRANS_DECODE
VAR_INPUT
	buffer : POINTER TO ARRAY[0..32000] OF BYTE;
END_VAR
VAR_IN_OUT
	length : DINT;
END_VAR
VAR_OUTPUT
	cmd : BOOL;
	device : STRING;
	key : STRING;
	error : BOOL;
END_VAR
VAR
	pt : POINTER TO BYTE;
	i : INT;
	stop : INT;
END_VAR

(*
	version 1.0	2 jan 2008
	programmer 	hugo
	tested BY		tobias

*)
(* do nothing if the buffer is empty *)
IF length > 0 THEN
	i := 0;
	error := TRUE;
	stop := DINT_TO_INT(length) - 2;
	(* read characters before first comma and store in device *)
	pt := ADR(device);
	WHILE i < stop DO
		IF buffer^[i] = 44 THEN EXIT; END_IF;
		pt^ := buffer^[i];
		pt := pt + 1;
		i := i + 1;
	END_WHILE;
	(* terminate the device string *)
	pt^ := 0;
	(* read after first comma and store in key *)
	i := i + 1;
	pt := ADR(key);
	WHILE i < stop DO
		pt^ := buffer^[i];
		pt := pt + 1;
		i := i + 1;
	END_WHILE;
	(* terminate the key string *)
	pt^:= 0;
	(* check if last two characters are $R$N 13, 10 *)
	IF buffer^[i] <> 13 AND buffer^[i+1] <> 10 THEN	RETURN;	END_IF;
	(* check if device and key are present *)
	IF LEN(device) = 0 OR LEN(key) = 0 THEN RETURN; END_IF;
	(* a valid transmission has been received *)
	cmd := TRUE;
	error := FALSE;
	(* clear the input buffer to allow the next transmission to occur *)
	length := 0;
ELSE
	error := FALSE;
	cmd := FALSE;
END_IF;


(* revision history
hm	2. jan 2008		rev 1.0
	original version

*)
END_FUNCTION_BLOCK

(* POU XTEST/Performance Test/measure_times, ST *)
FUNCTION_BLOCK measure_times
VAR_INPUT
END_VAR
VAR_OUTPUT
END_VAR
VAR
	times, mn, mx : ARRAY[0..300] OF REAL;
	tx: DWORD;
	init: BOOL;
	last: DWORD;
	t_max: DWORD := 100;
	cycles: DWORD;
	c_max: DWORD := 10000;
	i: INT;
	stop: INT := 9;
	overhead: REAL;
	runx : fc_list;
	timex: REAL;
END_VAR
IF NOT init THEN
	init := TRUE;
	_array_init(ADR(mn),SIZEOF(mn),99999);
END_IF;

IF i > stop THEN i := 0; END_IF;
(* measure overhead *)
last := TIME_TO_DWORD(TIME());
tx := 0;
cycles := 0;
WHILE tx < t_max AND cycles < c_max DO
	runx(num := i, check := TRUE);
	tx := TIME_TO_DWORD(TIME()) - last;
	cycles := cycles + 1;
END_WHILE;
overhead := DWORD_TO_REAL(tx) * 1000.0 / cycles;

(* measure execution time *)
last := TIME_TO_DWORD(TIME());
tx := 0;
cycles := 0;
WHILE tx < t_max AND cycles < c_max DO
	runx(num := i, check := FALSE);
	tx := TIME_TO_DWORD(TIME()) - last;
	cycles := cycles + 1;
END_WHILE;
timex := DWORD_TO_REAL(tx) * 1000.0 / cycles - overhead;

(* berechne korrekturwert für if anweisung für ckeck *)
IF i = 0 THEN
	mn[0] := MIN(timex,mn[0]);
	mx[0] := MAX(timex,mx[0]);
	times[0] := round((mx[0] + mn[0])/2,2);
ELSE
	mn[i] := MIN(timex - times[0], mn[i]);
	mx[i] := MAX(timex - times[0], mx[i]);
	times[i] := round((mx[i] + mn[i])/2,1);
END_IF;

i := i + 1;
END_FUNCTION_BLOCK

(* POU String/mirror, ST *)
FUNCTION mirror : STRING
VAR_INPUT
	str : STRING;
END_VAR
VAR
	pi : POINTER TO ARRAY[1..255] OF BYTE;
	po : POINTER TO BYTE;
	lx: INT;
	i: INT;
END_VAR

(*
version 1.0	4 feb 2008
programmer 	hugo
tested by		tobias

this function reverses an input string.

*)
pi := ADR(str);
po := ADR(mirror);
lx := LEN(str);
FOR i := lx TO 1 BY - 1 DO
	po^ := pi^[i];
	po := po + 1;
END_FOR;
(* close output string *)
po^:= 0;


(* revision histroy
hm		4. feb. 2008		rev 1.0
	original release

*)	
END_FUNCTION

(* POU other/Oscat_version, ST *)
FUNCTION Oscat_version : DWORD
VAR_INPUT
	in : BOOL;
END_VAR
VAR
END_VAR


(*
version 1.1	16 dec 2007
programmer 	hugo
tested by		tobias

oscat_version returns the version number in dword format
132 is library version 1.32
if IN = true then the release date will be returned

*)
IF in THEN
	Oscat_version := DATE_TO_DWORD(D#2008-2-11);
ELSE
	Oscat_version := 271;
END_IF;

(* revision history
hm	6. oct 2006	rev 1.0
	original version

hm	16. dec 2007	rev 1.1
	added possibility to return date and version depoending on in.
 
*)
END_FUNCTION

(* POU XTEST/Ideas/Ramp_S, ST *)
FUNCTION_BLOCK Ramp_S
VAR_INPUT
	X : REAL;
	KR : REAL;
	KF : REAL;
	A : REAL;
	RST : BOOL;
END_VAR
VAR_OUTPUT
	Y : REAL;
END_VAR
VAR
	speed : REAL;
	tx: DWORD;
	t_pls_ms: BOOL;
	last: DWORD;
	init: BOOL;
	phase: BYTE;
	in: BOOL;
	accelerate: BOOL;
END_VAR
(* read system time *)
IF NOT init OR rst THEN
	init := TRUE;
	Y := X;
ELSIF ABS(X - Y) > (speed * speed / A * 0.5) THEN
	accelerate := 0;
END_IF;
END_FUNCTION_BLOCK

(* POU engineering/signal processing/Range_to_Byte, ST *)
FUNCTION Range_to_Byte : BYTE
VAR_INPUT
	X : REAL;
	low : REAL;
	high : REAL;
END_VAR
VAR
END_VAR

(*
version 1.0	9. jan 2008
programmer 	hugo
tested by		tobias

Range_to_byte converts a real value between low and high into a byte

*)
Range_to_Byte := INT_TO_BYTE(TRUNC((LIMIT(low,X,high)-low) * 255.0 / (high - low)));


(* revision history
hm	9. jan 2008		rev 1.0
	original version

*)
END_FUNCTION

(* POU engineering/signal processing/Range_to_Word, ST *)
FUNCTION Range_to_Word : WORD
VAR_INPUT
	X : REAL;
	low : REAL;
	high : REAL;
END_VAR
VAR
END_VAR

(*
version 1.0	9. jan 2008
programmer 	hugo
tested by		tobias

Range_to_word converts a real value between low and high into a byte

*)
Range_to_Word := DINT_TO_WORD(TRUNC((LIMIT(low,X,high)-low) * 65535.0 / (high - low)));


(* revision history
hm	9. jan 2008		rev 1.0
	original version

*)
END_FUNCTION

(* POU XTEST/Baustein Tests/rdm_test, ST *)
FUNCTION_BLOCK rdm_test
VAR_INPUT
END_VAR
VAR_OUTPUT
END_VAR
VAR
	x: REAL;
	mx: REAL;
	Mn: REAL;
	x0, x1,x2, x3, x4, x5,x6, x7,x8, x9: REAL;
	V, U : REAL;
	W, G : REAL;
	C: DINT;
	CX0, cx1, cx2, cx3, cx4, cx5, cx6,cx7,cx8,cx9: REAL;
	CV: REAL;
	CU: REAL;
	CW : REAL;
	CG : REAL;
	last : ARRAY[0..11] OF REAL;
	sum : ARRAY[0..11] OF REAL;
	start: ARRAY[1..50] OF REAL;
	index: INT;
	sum1, sum2, sum3, sum4, sum5,sum6,sum7,sum8,sum9: REAL;
	last1, last2, last3, last4, last5, last6, last7, last8, last9: REAL;
	delta: REAL;
	d0, d1, d2, d3, d4, d5, d6,d7,d8,d9: REAL;
	dX0, dx1, dx2, dx3, dx4, dx5, dx6, dx7, dx8, dx9: REAL;
	d20, d21, d22, d23, d24, d25, d26,d27,d28,d29: REAL;
	dX20, dx21, dx22, dx23, dx24, dx25, dx26, dx27, dx28, dx29: REAL;
	oldtime: DWORD;
END_VAR
IF T_PLC_MS() = oldtime THEN RETURN; END_IF;
oldtime := T_PLC_MS();

C := c + 1;
x := RDM(x);
(* check if X is less then 0 or 1 or higher which is not allowed *)
IF X < 0 THEN Mn := mn +1;
ELSIF X >= 1 THEN mx := mx +1;

(* check distribution*)
ELSIF X < 0.1 THEN	x0 := x0+1; CX0 := C/10/x0;
ELSIF X < 0.2 THEN	x1 := x1+1; CX1 := C/10/x1;
ELSIF X < 0.3 THEN	x2 := x2+1; CX2 := C/10/x2;
ELSIF X < 0.4 THEN	x3 := x3+1; CX3 := C/10/x3;
ELSIF X < 0.5 THEN	x4 := x4+1; CX4 := C/10/x4;
ELSIF X < 0.6 THEN	x5 := x5+1; CX5 := C/10/x5;
ELSIF X < 0.7 THEN	x6 := x6+1; CX6 := C/10/x6;
ELSIF X < 0.8 THEN	x7 := x7+1; CX7 := C/10/x7;
ELSIF X < 0.9 THEN	x8 := x8+1; CX8 := C/10/x8;
ELSIF X < 1 THEN		x9 := x9+1; CX9 := C/10/x9;
END_IF;


(* check near 0 *)
IF X < 0.01 THEN V := V +1; END_IF; CV := C/100/V;
IF X < 0.001 THEN U := U +1; END_IF; CU := C/1000/U;

(* check near 1 *)
IF X >= 0.99 THEN W := W + 1; END_IF;CW := C/100/V;
IF X >= 0.999 THEN G := G + 1; END_IF; CG := C/1000/G;

(* check sequence1 *)
index := DINT_TO_INT(C MOD 12);
sum[index] := sum[index] + last[index] - X;
last[index] := X;

(* check sequence2 and delta to be distributed evenly *)
delta := last1 - X;
sum1 := sum1 + delta;
IF ABS(delta) < 0.1 THEN	d0 := d0+1; dX0 := C/10/d0;
ELSIF ABS(delta) < 0.2 THEN	d1 := d1+1; dX1 := C/10/d1;
ELSIF ABS(delta) < 0.3 THEN	d2 := d2+1; dX2 := C/10/d2;
ELSIF ABS(delta) < 0.4 THEN	d3 := d3+1; dX3 := C/10/d3;
ELSIF ABS(delta) < 0.5 THEN	d4 := d4+1; dX4 := C/10/d4;
ELSIF ABS(delta) < 0.6 THEN	d5 := d5+1; dX5 := C/10/d5;
ELSIF ABS(delta) < 0.7 THEN	d6 := d6+1; dX6 := C/10/d6;
ELSIF ABS(delta) < 0.8 THEN	d7 := d7+1; dX7 := C/10/d7;
ELSIF ABS(delta) < 0.9 THEN	d8 := d8+1; dX8 := C/10/d8;
ELSIF ABS(delta) < 1 THEN   d9 := d9+1; dX9 := C/10/d9;
END_IF;
last1 := X;


IF c MOD 2 = 0 THEN
	delta := last2 - X;
	sum2 := sum2 + delta;
	IF ABS(delta) < 0.1 THEN	d20 := d20+1; dX20 := C/20/d20;
	ELSIF ABS(delta) < 0.2 THEN	d21 := d21+1; dX21 := C/20/d21;
	ELSIF ABS(delta) < 0.3 THEN	d22 := d22+1; dX22 := C/20/d22;
	ELSIF ABS(delta) < 0.4 THEN	d23 := d23+1; dX23 := C/20/d23;
	ELSIF ABS(delta) < 0.5 THEN	d24 := d24+1; dX24 := C/20/d24;
	ELSIF ABS(delta) < 0.6 THEN	d25 := d25+1; dX25 := C/20/d25;
	ELSIF ABS(delta) < 0.7 THEN	d26 := d26+1; dX26 := C/20/d26;
	ELSIF ABS(delta) < 0.8 THEN	d27 := d27+1; dX27 := C/20/d27;
	ELSIF ABS(delta) < 0.9 THEN	d28 := d28+1; dX28 := C/20/d28;
	ELSIF ABS(delta) < 1 THEN   d29 := d29+1; dX29 := C/20/d29;
	END_IF;
	last2 := X;
END_IF;
IF c MOD 3 = 0 THEN
	sum3 := sum3 + last3 - x; last3 := X;
END_IF;
IF c MOD 4 = 0 THEN
	sum4 := sum4 + last4 - x; last4 := X;
END_IF;
IF c MOD 5 = 0 THEN
	sum5 := sum5 + last5 - x; last5 := X;
END_IF;
IF c MOD 6 = 0 THEN
	sum6 := sum6 + last6 - x; last6 := X;
END_IF;
IF c MOD 7 = 0 THEN
	sum7 := sum7 + last7 - x; last7 := X;
END_IF;
IF c MOD 8 = 0 THEN
	sum8 := sum8 + last8 - x; last8 := X;
END_IF;
IF c MOD 9 = 0 THEN
	sum9 := sum9 + last9 - x; last9 := X;
END_IF;

(* store startup sequence *)
IF c <= 50 THEN
	start[DINT_TO_INT(C)] := X;
END_IF;
END_FUNCTION_BLOCK

(* POU String/REPLACE_ALL, ST *)
FUNCTION REPLACE_ALL : STRING
VAR_INPUT
	str : STRING;
	src : STRING;
	rep : STRING;
END_VAR
VAR
	pos: INT;
	lp : INT;
	lx : INT;
END_VAR

(*
version 1.0	4 feb 2008
programmer 	hugo
tested by		tobias

the function findP searches a string str for the occurence of src beginning at the position pos.

*)
REPLACE_ALL := str;
lx := LEN(src);
lp := LEN(rep);
pos := FINDP(REPLACE_ALL, src, 1);
WHILE pos > 0 DO
	REPLACE_ALL := REPLACE(REPLACE_ALL,rep,lx, pos);
	pos := FINDP(REPLACE_ALL, src, pos + lp);
END_WHILE;

(* revision histroy
hm		4. feb. 2008		rev 1.0
	original release

*)	
END_FUNCTION

(* POU Time&Date/RTC_2, ST *)
FUNCTION_BLOCK RTC_2
VAR_INPUT
	SET : BOOL;
	SDT : DT;
	SMS : INT;
	DEN : BOOL;
	OFS : INT;
END_VAR
VAR_OUTPUT
	UDT : DT;
	LDT : DT;
	DSO : BOOL;
	XMS : INT;
END_VAR
VAR
	RT : RTC_MS;
	T: INT;
END_VAR

(*
version 1.1	20. feb. 2008
programmer 	hugo
tested by	tobias

RTC_2 is a real time clock module which runs utc and generates local time from utc.
daylight savings time can be enabled with den and an additional local time is generated with a delay of ofs.

*)
(* call rtc *)
RT(SET := SET, SDT := SDT, SMS := SMS);
UDT := rt.xdt;
XMS := rt.XMS;

(* check for daylight savings time and set dso output *)
dso := DST(udt) AND DEN;
IF dso THEN T := 1; ELSE T := 0; END_IF;

(* calculate time offset and set ldt output *)
LDT := DWORD_TO_DT(DT_TO_DWORD(UDT) + INT_TO_DWORD(ofs + T) * 3600);


(* revision history
hm		20. jan. 2008	rev 1.0
	original version

hm		20. feb. 2008	rev 1.1
	added Millisecond Set input
*)
END_FUNCTION_BLOCK

(* POU Time&Date/RTC_MS, ST *)
FUNCTION_BLOCK RTC_MS
VAR_INPUT
	SET : BOOL;
	SDT : DT;
	SMS : INT;
END_VAR
VAR_OUTPUT
	XDT : DT;
	XMS : INT;
END_VAR
VAR
	init: BOOL;
	last: DWORD;
	Tx: DWORD;
END_VAR

(*
version 1.1	20. feb. 2008
programmer 	hugo
tested by	tobias

RTC_MS is a real time clock module which can be set to SDT when set is TRUE and the outputs XDT and XT present the DateTime and TOD with a resolution of milliseconds.

*)
tx := T_PLC_MS();
IF set OR NOT init THEN
	(* clock needs to be set when set is true or after power up *)
	init := TRUE;
	xdt := SDT;
	XMS := SMS;
ELSE
	XMS := XMS + DWORD_TO_INT(tx - last);
	(* check if one second has expired *)
	IF XMS > 999 THEN
		XDT := XDT + T#1s;
		XMS := XMS - 1000;
	END_IF;
END_IF;
last := tx;


(* revision history
hm		20. jan. 2008	rev 1.0
	original version

hm		20. feb. 2008	rev 1.1
	added Millisecond Set input
*)
END_FUNCTION_BLOCK

(* POU Logic/FF edge triggered/select_8, ST *)
FUNCTION_BLOCK select_8
VAR_INPUT
	EN : BOOL;
	SET : BOOL;
	IN : BYTE;
	UP : BOOL;
	DN : BOOL;
	RST : BOOL;
END_VAR
VAR_OUTPUT
	Q0, Q1, Q2, Q3, Q4, Q5, Q6, Q7 : BOOL;
		STATE : INT;
END_VAR
VAR
	last_up: BOOL;
	last_dn : BOOL;
END_VAR

(*
	version 1.0	16 jan 2008
	programmer 	hugo
	tested BY	tobias

select_8 selects one of 8 outputs at any time. the outputscan be selected by up or down keys and an independent anable switches all outouts off if set false


*)
IF rst THEN
	state := 0;
ELSIF set THEN
	state := IN;
ELSIF up AND NOT last_up THEN
	state := inc(state,1,7);
ELSIF dn AND NOT last_dn THEN
	state := inc(state,-1,7);
END_IF;
last_UP := UP;
last_DN := DN;

Q0 := FALSE;
Q1 := FALSE;
Q2 := FALSE;
Q3 := FALSE;
Q4 := FALSE;
Q5 := FALSE;
Q6 := FALSE;
Q7 := FALSE;

IF en THEN
	CASE state OF
		0: Q0 := TRUE;
		1: Q1 := TRUE;
		2: Q2 := TRUE;
		3: Q3 := TRUE;
		4: Q4 := TRUE;
		5: Q5 := TRUE;
		6: Q6 := TRUE;
		7: Q7 := TRUE;
	END_CASE;
END_IF;

(* revision history
hm	16. jan 2008	rev 1.0
	original version

*)
END_FUNCTION_BLOCK

(* POU XTEST/Baustein Tests/set_date_test, ST *)
FUNCTION_BLOCK set_date_test
VAR_INPUT
END_VAR
VAR_OUTPUT
	OK : BOOL;
	rx : DWORD;
	fdate : DATE;
END_VAR
VAR
	yr : INT;
	last: REAL;
	day: INT;
	i: INT;
	temp: DATE;
	init: BOOL;
	mth: INT;
END_VAR
IF NOT init THEN
	ok := TRUE;
	init := TRUE;
END_IF;
FOR i := 1 TO 1000 DO
	last := RDM(last);
	yr := TRUNC(last * 130 + 1970);
	last := RDM(last);
	mth := TRUNC(last * 11.999) + 1;
	last := RDM(last);
	day := TRUNC(last * 30.999) + 1;
	CASE mth OF
		2 : IF leap_year(yr) THEN IF day > 29 THEN day := 29; END_IF;	ELSE IF day > 28 THEN day := 28; END_IF; END_IF;
		4 : IF day > 30 THEN day := 30; END_IF;
		6 : IF day > 30 THEN day := 30; END_IF;
		9 : IF day > 30 THEN day := 30; END_IF;
		11 : IF day > 30 THEN day := 30; END_IF;
	END_CASE;
	temp := set_Date(yr,mth,day);
	IF month(temp) <> mth THEN
		ok := FALSE;
		fdate := temp;
	END_IF;
	IF year(temp) <> yr THEN
		ok := FALSE;
		fdate := temp;
	END_IF;
	IF day_of_month(temp) <> day THEN
		ok := FALSE;
		fdate := temp;
	END_IF;
	rx := rx + 1;
END_FOR;
END_FUNCTION_BLOCK

(* POU XTEST/Ideas/sntp, ST *)
FUNCTION_BLOCK sntp
VAR_INPUT
	SET : BOOL;
END_VAR
VAR_OUTPUT
	TP :	BOOL;
	UDT :	UDINT;
	XMS :	INT;
	error :	BOOL;
END_VAR
(*
VAR_IN_OUT
	xStartSend :	BOOL;
	snd_length :	DINT;
	snd_buffer :	oscat_us_IP_DATA;
	rec_length :	DINT;
	rev_buffer :	oscat_us_IP_DATA;
END_VAR
VAR
	i :	INT;
	state :	INT;
	last :	UDINT;
	tx :	UDINT;
END_VAR *)
RETURN;
(*
(* read system time *)
tx := T_PLC_MS();

CASE state OF

00: (* Domain Name System (query) *)
  IF SET = FALSE THEN RETURN; END_IF;

  snd_buffer.bya_IP_DATA[01] := BYTE#16#1B;
  FOR i := 2 TO 48 DO
    snd_buffer.bya_IP_DATA[i] := BYTE#16#00;
  END_FOR;

  snd_length := DINT#48;
  xStartSend := TRUE;  
  state := 01;
  TP := FALSE;
  error := FALSE;
  last := tx;

01:
  (* Receive Data - Timeout 6 sek. *)
  IF (tx - last) > UDINT#6000 THEN
    snd_length := DINT#00;
    state := 3;
    error := TRUE; (* Timeout *)
  END_IF;
  
  (* länge der empfangenen Daten prüfen *)
  IF rec_length  < DINT#48 THEN RETURN; END_IF;

  (* Umrechnung SNTP Timestamp Base 1900-01-01 mit Internet Byte-Order -> Unix 1970-01-01 = +2208988800 sekunden*)
  UDT := DWORD_TO_UDINT(DWord_of_Byte(rev_buffer.bya_IP_DATA[44],rev_buffer.bya_IP_DATA[43],rev_buffer.bya_IP_DATA[42],rev_buffer.bya_IP_DATA[41]))- UDINT#2208988800;

  (* Original-Sekundenanteile sind als 32 Bit Fractal dargestellt *) 
  (* ms nur mit veringerte Auflösung berechnen 1/65535 -> Highword verwenden *)

  (* schnelle Version: durch 64 dividieren -> führt zu ca 25ms Rechenfehler *)
  XMS := WORD_TO_INT(SHR_WORD(Word_of_Byte(rev_buffer.bya_IP_DATA[46],rev_buffer.bya_IP_DATA[45]),6));

  (* genauere Variante noch besser wäre / REAL#65.535 aber ......... 
  XMS := UINT_TO_INT(WORD_TO_UINT(Word_of_Byte(rev_buffer.bya_IP_DATA[46],rev_buffer.bya_IP_DATA[45])) / UINT#66);
  *)

  (* Zeitdifferenz (Laufzeitfehler) zwischen Send und Receive /2 teilen *)
  XMS := XMS + DWORD_TO_INT(SHR_DWORD(UDINT_TO_DWORD(tx - last),1));

  (* sekundenanteile der Zeitdifferenz *)
  UDT := UDT + INT_TO_UDINT(XMS / 1000);
  (* ms übernehmen *)
  XMS := XMS MOD 1000;

  snd_length := DINT#00;
  state := 2;
  TP := TRUE;

02:
  TP := FALSE;
  
  IF SET = FALSE THEN 
    state := 0;
    error := FALSE;
  END_IF;
END_CASE;

(*               SNTP Datenstruktur
                                  1                   2                   3
              0 1 2 3 4 5 6 7 8 9 0 1 2 3 4 5 6 7 8 9 0 1 2 3 4 5 6 7 8 9 0 1
             +-+-+-+-+-+-+-+-+-+-+-+-+-+-+-+-+-+-+-+-+-+-+-+-+-+-+-+-+-+-+-+-+
Byte: 01-04  |LI | VN  |Mode |    Stratum    |     Poll      |   Precision   |
             +-+-+-+-+-+-+-+-+-+-+-+-+-+-+-+-+-+-+-+-+-+-+-+-+-+-+-+-+-+-+-+-+
Byte: 05-08  |                          Root  Delay (32 Bit)                 |
             +-+-+-+-+-+-+-+-+-+-+-+-+-+-+-+-+-+-+-+-+-+-+-+-+-+-+-+-+-+-+-+-+
Byte: 09-12  |                       Root  Dispersion (32 Bit)               |
             +-+-+-+-+-+-+-+-+-+-+-+-+-+-+-+-+-+-+-+-+-+-+-+-+-+-+-+-+-+-+-+-+
Byte: 13-16  |                     Reference Identifier (32 Bit)             |
             +-+-+-+-+-+-+-+-+-+-+-+-+-+-+-+-+-+-+-+-+-+-+-+-+-+-+-+-+-+-+-+-+
Byte: 17-24  |                    Reference Timestamp (64 Bit)               |
             +-+-+-+-+-+-+-+-+-+-+-+-+-+-+-+-+-+-+-+-+-+-+-+-+-+-+-+-+-+-+-+-+
Byte: 25-32  |                    Originate Timestamp (64 Bit)               |
             +-+-+-+-+-+-+-+-+-+-+-+-+-+-+-+-+-+-+-+-+-+-+-+-+-+-+-+-+-+-+-+-+
Byte: 33-40  |                     Receive Timestamp (64 Bit)                |
             +-+-+-+-+-+-+-+-+-+-+-+-+-+-+-+-+-+-+-+-+-+-+-+-+-+-+-+-+-+-+-+-+
Byte: 41-48  |                     Transmit Timestamp (64 Bit)               |
             +-+-+-+-+-+-+-+-+-+-+-+-+-+-+-+-+-+-+-+-+-+-+-+-+-+-+-+-+-+-+-+-+
Byte: 49-52  |                 Key Identifier (optional) (32 Bit)            |
             +-+-+-+-+-+-+-+-+-+-+-+-+-+-+-+-+-+-+-+-+-+-+-+-+-+-+-+-+-+-+-+-+
Byte: 53-68  |                 Message Digest (optional) (128 Bit)           |
             +-+-+-+-+-+-+-+-+-+-+-+-+-+-+-+-+-+-+-+-+-+-+-+-+-+-+-+-+-+-+-+-+

*)

(*
Worldwide NTP-Server


NIST-Zeitserver
• time-a.nist.gov
129.6.15.28 
NIST, Gaithersburg, Maryland 
• time-a.nist.gov
129.6.15.28 
NIST, Gaithersburg, Maryland 
• time-a.timefreq.bldrdoc.gov
132.163.4.101 (Stand: 1. Dezember 1999)
NIST, Boulder, Colorado 
• time-b.timefreq.bldrdoc.gov
132.163.4.102 (Stand: 1. Dezember 1999)
NIST, Boulder, Colorado 
• time-c.timefreq.bldrdoc.gov
132.163.4.103 (Stand: 1. Dezember 1999)
NIST, Boulder, Colorado 
• utcnist.colorado.edu
128.138.140.44
University of Colorado, Boulder 
• time.nist.gov
192.43.244.18
NCAR, Boulder, Colorado 
• time-nw.nist.gov
131.107.1.10
Microsoft, Redmond, Washington 
• nist1.dc.certifiedtime.com
216.200.93.8
Abovnet, North Virginia 
• nist1.datum.com
209.0.72.7
Datum, San Jose, Kalifornien 
• nist1.nyc.certifiedtime.com
208.184.49.129 
Abovnet, New York City 
• nist1.sjc.certifiedtime.com
207.126.103.202
Abovnet, San Jose, Kalifornien 

Zeitserver der ersten Ebene
Sortiert nach Standort: 
Nordamerika
• Palo Alto, Kalifornien: Systems Research Center, Compaq Computer Corp.
204.123.2.72: usno.pa-x.dec.com; CNAME: navobs1.pa-x.dec.com
Servicebereich: US-Zeitzonen PST (Pacific Standard Time) und MST (Mountain Standard Time) 
• Marina del Rey, Kalifornien: USC Information Sciences Institute
128.9.176.30: timekeeper.isi.edu
Servicebereich: CalRen2- und Los Nettos-Bereich  
• Washington, DC: U.S. Naval Observatory
192.5.41.41: tock.usno.navy.mil 
192.5.41.40: tick.usno.navy.mil
Servicebereich: NSFNET 
• Ottawa, Ontario, Kanada: National Research Council of Canada
time.chu.nrc.ca
Servicebereich: Kanada 
• Raleigh, North Carolina: North Carolina State University
152.1.58.124: terrapin.csc.ncsu.edu
Servicebereich: Südosten der USA 
• Cambridge, Massachusetts: MIT Information Systems
18.72.0.3: bitsy.mit.edu 
Servicebereich: NSFNET- und NEARnet-Bereich 
• Cambridge, Massachusetts: MIT
18.26.4.105: bonehed.lcs.mit.edu
Servicebereich: Osten der USA 
• Palo Alto, Kalifornien: Internet Software Consortium
192.5.5.250: clock.isc.org
Servicebereich: BARRnet, Alternet-West und CIX-West 
• Cambridge, Massachusetts: Open Software Foundation
130.105.4.59: clock.osf.org
Servicebereich: NSFNET- und NEARnet-Bereich 
• Palo Alto, Kalifornien: ViaNet Communications
209.81.9.7: clock.via.net 
• Cleveland, Ohio: Lewis Research Center (NASA)
128.156.1.43: lerc-dns.lerc.nasa.gov
Servicebereich: NSFNET und OARNET 
• Colorado Springs, Colorado: Schriever AFB
204.34.198.40: navobs1.usnogps.navy.mil; CNAME: tick.usnogps.navy.mil 
204.34.198.41: navobs1.usnogps.navy.mil; CNAME: tock.usnogps.navy.mil 
Servicebereich: US-Zeitzonen PST (Pacific Standard Time) und MST (Mountain Standard Time) 
• St. Louis, Missouri: Washington University
128.252.19.1: navobs1.usnogps.navy.mil; CNAME: tick.wustl.edu 
Servicebereich: US-Zeitzone CST (Central Standard Time) 
• Research Triangle Park, North Carolina: MCNC
192.101.21.1: ncnoc.ncren.net
Servicebereich: NC-REN-Bereich (North Carolina Research and Education Network) 
• Cupertino, Kalifornien: HP
192.6.38.127: ntp-cup.external.hp.com
Servicebereich: USA Westküste 
• Newark, Delaware: Conectiv Communications
138.39.7.20: ntp1.delmarva.com
Servicebereich: Cable & Wireless Network (früher MCInet) 
• University Park, Pennsylvania: Penn State University
128.118.46.3: otc1.psu.edu
Servicebereich: NSFNET, PREPNET und JvNCnet  

Europa
• Borowiec, Polen: Astrogeodynamical Observatory, Space Research Centre
150.254.183.15: vega.cbk.poznan.pl
Servicebereich: Polen und Europa 
• Stockholm, Schweden: Stupi AB
192.36.143.151: Time2.Stupi.SE
Servicebereich: Europa 
• Turin, Italien: IEN Galileo Ferraris
193.204.114.1: time.ien.it
Servicebereich: Italien und Europa 
• Zürich, Schweiz: Integrated Systems Laboratory , Eidgenössischen Technischen Hochschule Zürich 
129.132.2.21: swisstime.ethz.ch
Servicebereich: Schweiz und Europa 
• Turin, Italien: CSTV of National Research Council
150.145.33.1: tempo.cstv.to.cnr.it
Servicebereich: Italien und Europa 
• Erlangen, Deutschland: Universität Erlangen-Nürnberg
ntp0.fau.de; ntp1.fau.de; ntp2.fau.de; 
ntps1-0.uni-erlangen.de; ntps1-1.uni-erlangen.de; ntps1-2.uni-erlangen.de
Servicebereich: Deutschland und Europa 
• Berlin, Deutschland: Technische Universität Berlin
130.149.17.21: ntps1-0.cs.tu-berlin.de
130.149.17.8: ntps1-1.cs.tu-berlin.de
Servicebereich: Deutschland und Europa 
• Deutschland
131.173.17.7: ntps1-1.rz.Uni-Osnabrueck.DE
Servicebereich: Deutschland und Europa 
• Schweden
192.36.143.150: Time1.Stupi.SE
Servicebereich: SUnet und NORDUnet Schweden 

Fernost und pazifische Randgebiete
• Hong Kong: Chinesische Universität von Hong Kong. 
137.189.6.18: clock.cuhk.edu.hk
Servicebereich: Hong Kong (China) und Südostasien  
• Fukuoka, Japan: Universität Fukuoka
133.100.9.2: clock.nc.fukuoka-u.ac.jp
133.100.11.8: clock.tl.fukuoka-u.ac.jp
Servicebereich: Japan und pazifischer Raum  

Australien
• Melbourne, Australien: University of Melbourne
128.250.36.2: ntp.cs.mu.OZ.AU
Servicebereich: Australien und Neuseeland  

Zeitserver der zweiten Ebene
Nach geographischem Standort sortiert: 
Nordamerika
NTP-Zeitserver: • Quebec, Kanada: Canadian Meteorological Center
ntp1.cmc.ec.gc.ca; ntp2.cmc.ec.gc.ca 
Servicebereich: Ostkanada  
• Ontario, Kanada: National Research Council of Canada
time.chu.nrc.ca; time.nrc.ca
Servicebereich: Kanada 
• Saskatchewan, Kanada: University of Regina 
142.3.100.15: timelord.uregina.ca
Servicebereich: Kanada 
• Ontario, Kanada: University of Toronto
tick.utoronto.ca; tock.utoronto.ca
Servicebereich: Ostkanada  
• Mexiko: Audiotel-Büro 
ntp2a.audiotel.com.mx; ntp2c.audiotel.com.mx; ntp2b.audiotel.com.mx
Servicebereich: Avantel, MCINet und Mexiko 
• Santa Cruz, Kalifornien: Scruz-net, inc.
165.227.1.1: ns.scruz.net
Servicebereich: Westen der USA 
• San Diego, Kalifornien: UCSD Academic Computing Services/Network Operations
132.239.254.49: ntp.ucsd.edu
Servicebereich: CERFNET; NSFNET, SDSC-Bereich, und nahegelegene Bereiche 
• Quincy, Kalifornien 
ntp1.mainecoon.com; ntp2.mainecoon.com 
Servicebereich: Nordamerika 
• Newark, Delaware: University of Delaware
128.175.1.3: louie.udel.edu
Servicebereich: CAIRN, Abilene und vBNS  
• Atlanta, Georgia: CNSG
ntp.shorty.com
Servicebereich: Südwesten der USA  
• Kennesaw, Georgia: PeachNet 
rolex.peachnet.edu; timex.peachnet.edu
Servicebereich: PeachNet (Georgia) und Südwesten der USA  
• Urbana-Champaign, Illinois: University of Illinois
ntp-0.cso.uiuc.edu; ntp-1.cso.uiuc.edu; ntp-2.cso.uiuc.edu
Servicebereich: CICNET, Mittlerer Westen und NCSA-Bereich  
• Chicago, Illinois: Argonne National Laboratory 
ntp-1.mcs.anl.gov; ntp-2.mcs.anl.gov
Servicebereich: NSF/ANSNet, CICNet, NetIllinois und ESNet  
• West Lafayette, Indiana: Purdue University
gilbreth.ecn.purdue.edu; harbor.ecn.purdue.edu; molecule.ecn.purdue.edu 
Servicebereich: NSFNET- und CICNET-Bereich  
• Manhattan, Kansas: KansasNet OnLine Services
199.240.130.1: ntp1.kansas.net
199.240.130.12: ntp2.kansas.net
Servicebereich: Zentral-USA und Great Plains  
• Boston, Massachusetts: UMass-Boston CS dept.
158.121.104.4: timeserver.cs.umb.edu
Servicebereich: Neuengland  
• Minneapolis/St Paul, Minnesota: University of Minnesota
ns.nts.umn.edu; nss.nts.umn.edu
Servicebereich: CICNET-Bereich  
• Columbia, Missouri: University of Missouri-Columbia
128.206.206.12: everest.cclabs.missouri.edu
Servicebereich: MOREnet  
• Omaha, Nebraska: Radiks Internet Access
205.138.126.83: allison.radiks.net
Servicebereich: Mittlerer Westen, USA  
• Las Vegas, Nevada: University of Nevada System Computing Services
131.216.1.101: cuckoo.nevada.edu 
Servicebereich: NevadaNet, NSFNET und SDSC-Bereich  
• Las Vegas, Nevada: UNLV College of Engineering
tick.cs.unlv.edu; tock.cs.unlv.edu
Servicebereich: Sprintnet  
• New York City, New York: Columbia University
ntp.ctr.columbia.edu 
Servicebereich: Sprintlink und NYSERnet  
• Ithaca, New York: Cornell University 
192.35.82.50: ntp0.cornell.edu
Servicebereich: NSFNET und NYSER-Bereich  
• New York, New York: Morningside Campus, Columbia University
sundial.columbia.edu
Servicebereich: NYSERnet  
• New York City, New York: Columbia University Computer Science Department
timex.cs.columbia.edu 
Servicebereich: PSINET; NSFNET, und NYSER-Bereich  
• Norman, Oklahoma: University of Oklahoma
129.15.22.8: constellation.ecn.uoknor.edu 
Servicebereich: Midnet  
• Coos Bay, Oregon: Koala Computers
207.48.109.6: tick.koalas.com
Servicebereich: Nordwesten der USA  
• University Park, Pennsylvania: Penn State University
128.118.25.3: clock.psu.edu
Servicebereich: Internet2, vBNS, CERFnet(AT&T IP Services), PSC/NCNE und CASC 
• Pittsburgh, Pennsylvania: Pittsburgh Supercomputing Center
128.182.58.100: fuzz.psc.edu
Servicebereich: NSFNET und PSC-Bereich  
• Pittsburgh, Pennsylvania: Carnegie Mellon Electrical and Computer Engineering 
ntp-1.ece.cmu.edu; ntp-2.ece.cmu.edu 
Servicebereich: PREPNET und PSC-Bereich  
• Dallas, Texas: Cox School of Business, Southern Methodist University
129.119.80.126: ntp.cox.smu.edu 
Servicebereich: NSFNET und SESQUI-Bereich  
• Hughes Springs, Texas: First National Bank
209.144.20.76: ntp.fnbhs.com
Servicebereich: Nordosten Texas  
• Houston, Texas: Baylor College of Medicine
128.249.1.10: ntp.tmc.edu 
Servicebereich: NSFNET und SESQUI-Bereich  
• College Station, Texas: Texas A&M University
165.91.52.110: ntp5.tamu.edu
Servicebereich: NSFNET, SESQUI-Bereich, THEnet und TAMUSDSN 
• Plano, Texas: Greyware Automation Products
tick.greyware.com; tock.greyware.com
Servicebereich: Südzentral-USA  
• Blacksburg, Virginia: Virginia Tech Computing Center
ntp-1.vt.edu; ntp-2.vt.edu
Servicebereich: Südwesten der USA  
• Arlington, Virginia: Center for Seismic Studies
140.162.1.3: ntp.cmr.gov
Servicebereich: NSFNET und SURA-Bereich  
• Richland, Washington: Washington State University 
192.31.216.30: clock.tricity.wsu.edu
Servicebereich: NSFNET und NorthWestNet  
• Washington, USA: Mill Creek
time.ultimeth.net
Servicebereich: Nordwesten der USA  
• Wisconsin, USA: Computer Science Department, University of Wisconsin-Madison
ntp1.cs.wisc.edu; ntp2.cs.wisc.edu; ntp3.cs.wisc.edu
Servicebereich: USA und jeder andere  

Südamerika
• Buenos Aires, Argentinien: Network Access Point
200.49.40.1: CNAME: tick.nap.com.ar
200.49.32.1: CNAME: tock.nap.com.ar
Servicebereich: Argentinien 
• Buenos Aires, Argentinien: Sinectis S.A.
time.sinectis.com.ar 
Servicebereich: Argentinien 
• Brasilien: Brazilian Research Network
200.144.121.33: ntp.cais.rnp.br 
Servicebereich: Brasilien 
• Venezuela: VELUG, Grupo de Usuarios Linux de Venezuela
150.185.192.250: ntp.linux.org.ve
Servicebereich: Arica  

